// Mitsubishi GX Works2 project: A02_20260228_0   PLC: Q03UDV

TYPE Auto_Data : STRUCT
  X軸現在位置 : REAL;
  Y軸現在位置 : REAL;
END_STRUCT END_TYPE

// global labels: Global1
VAR_GLOBAL
  Auto_Data : Auto_Data;
  現在位置列 AT D400 : INT;
  現在位置層 AT D402 : INT;
END_VAR

// global labels: Coords
VAR_GLOBAL
  列座標 AT D3284 : ARRAY [1..14] OF REAL;
  層座標 AT D3274 : ARRAY [1..5] OF REAL;
  Z座標 AT D3270 : ARRAY [1..2] OF REAL;
END_VAR

PROGRAM 09  // Alram
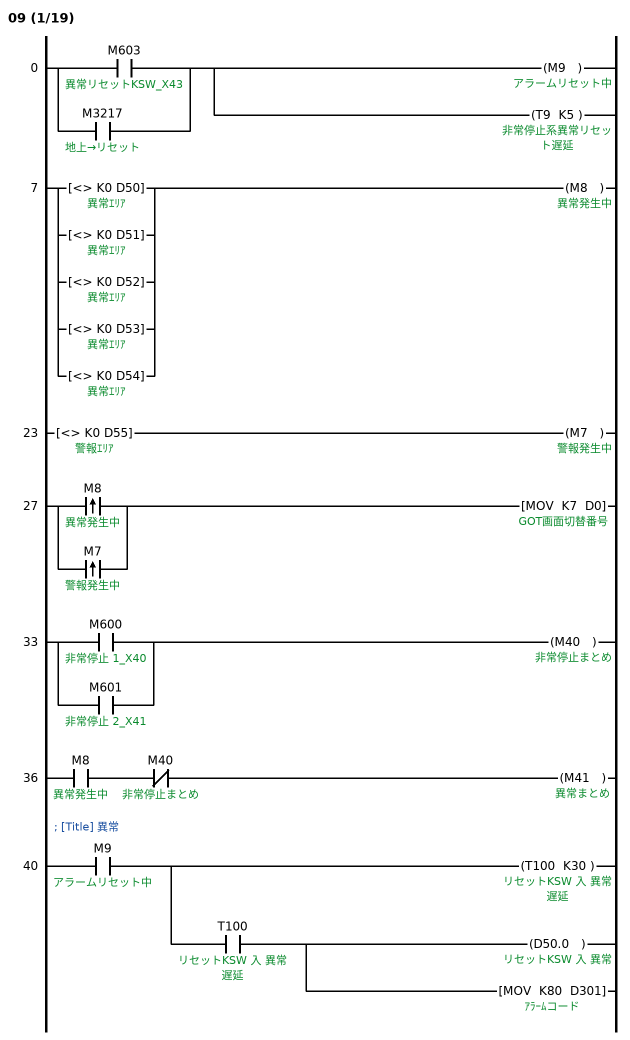
0     LD      M603  ; 異常リセットKSW_X43
      OR      M3217  ; 地上→リセット
      OUT     M9  ; アラームリセット中
      OUT     T9 K5  ; 非常停止系異常リセット遅延
7     LD<>    K0 D50  ; 異常ｴﾘｱ
      OR<>    K0 D51  ; 異常ｴﾘｱ
      OR<>    K0 D52  ; 異常ｴﾘｱ
      OR<>    K0 D53  ; 異常ｴﾘｱ
      OR<>    K0 D54  ; 異常ｴﾘｱ
      OUT     M8  ; 異常発生中
23    LD<>    K0 D55  ; 警報ｴﾘｱ
      OUT     M7  ; 警報発生中
27    LDP     M8  ; 異常発生中
      ORP     M7  ; 警報発生中
      MOV     K7 D0  ; GOT画面切替番号
33    LD      M600  ; 非常停止 1_X40
      OR      M601  ; 非常停止 2_X41
      OUT     M40  ; 非常停止まとめ
36    LD      M8  ; 異常発生中
      ANI     M40  ; 非常停止まとめ
      OUT     M41  ; 異常まとめ
; [Title] 異常
40    LD      M9  ; アラームリセット中
      OUT     T100 K30  ; リセットKSW 入 異常 遅延
      AND     T100  ; リセットKSW 入 異常 遅延
      OUT     D50.0  ; リセットKSW 入 異常
      MOV     K80 D301  ; ｱﾗｰﾑコード
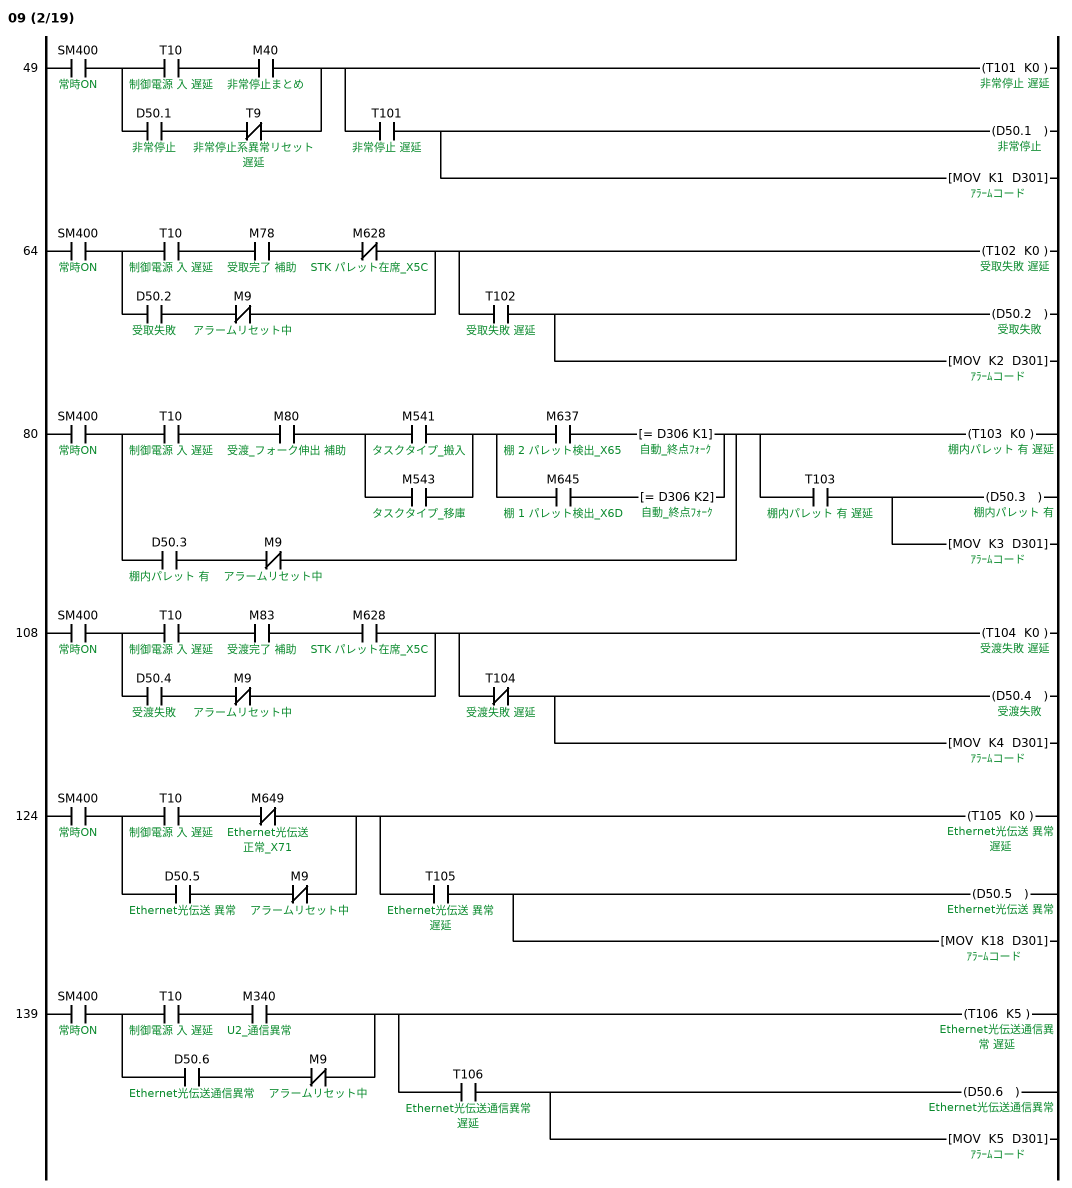
49    LD      SM400  ; 常時ON
      LD      T10  ; 制御電源 入 遅延
      AND     M40  ; 非常停止まとめ
      LD      D50.1  ; 非常停止
      ANI     T9  ; 非常停止系異常リセット遅延
      ORB
      ANB
      OUT     T101 K0  ; 非常停止 遅延
      AND     T101  ; 非常停止 遅延
      OUT     D50.1  ; 非常停止
      MOV     K1 D301
64    LD      SM400  ; 常時ON
      LD      T10  ; 制御電源 入 遅延
      AND     M78  ; 受取完了 補助
      ANI     M628  ; STK パレット在席_X5C
      LD      D50.2  ; 受取失敗
      ANI     M9  ; アラームリセット中
      ORB
      ANB
      OUT     T102 K0  ; 受取失敗 遅延
      AND     T102  ; 受取失敗 遅延
      OUT     D50.2  ; 受取失敗
      MOV     K2 D301
80    LD      SM400  ; 常時ON
      LD      T10  ; 制御電源 入 遅延
      AND     M80  ; 受渡_フォーク伸出 補助
      LD      M541  ; タスクタイプ_搬入
      OR      M543  ; タスクタイプ_移庫
      ANB
      LD      M637  ; 棚 2 パレット検出_X65
      AND=    D306 K1  ; 自動_終点ﾌｫｰｸ
      LD      M645  ; 棚 1 パレット検出_X6D
      AND=    D306 K2  ; 自動_終点ﾌｫｰｸ
      ORB
      ANB
      LD      D50.3  ; 棚内パレット 有
      ANI     M9  ; アラームリセット中
      ORB
      ANB
      OUT     T103 K0  ; 棚内パレット 有 遅延
      AND     T103  ; 棚内パレット 有 遅延
      OUT     D50.3  ; 棚内パレット 有
      MOV     K3 D301
108   LD      SM400  ; 常時ON
      LD      T10  ; 制御電源 入 遅延
      AND     M83  ; 受渡完了 補助
      AND     M628  ; STK パレット在席_X5C
      LD      D50.4  ; 受渡失敗
      ANI     M9  ; アラームリセット中
      ORB
      ANB
      OUT     T104 K0  ; 受渡失敗 遅延
      ANI     T104  ; 受渡失敗 遅延
      OUT     D50.4  ; 受渡失敗
      MOV     K4 D301
124   LD      SM400  ; 常時ON
      LD      T10  ; 制御電源 入 遅延
      ANI     M649  ; Ethernet光伝送 正常_X71
      LD      D50.5  ; Ethernet光伝送 異常
      ANI     M9  ; アラームリセット中
      ORB
      ANB
      OUT     T105 K0  ; Ethernet光伝送 異常 遅延
      AND     T105  ; Ethernet光伝送 異常 遅延
      OUT     D50.5  ; Ethernet光伝送 異常
      MOV     K18 D301
139   LD      SM400  ; 常時ON
      LD      T10  ; 制御電源 入 遅延
      AND     M340  ; U2_通信異常
      LD      D50.6  ; Ethernet光伝送通信異常
      ANI     M9  ; アラームリセット中
      ORB
      ANB
      OUT     T106 K5  ; Ethernet光伝送通信異常 遅延
      AND     T106  ; Ethernet光伝送通信異常 遅延
      OUT     D50.6  ; Ethernet光伝送通信異常
      MOV     K5 D301
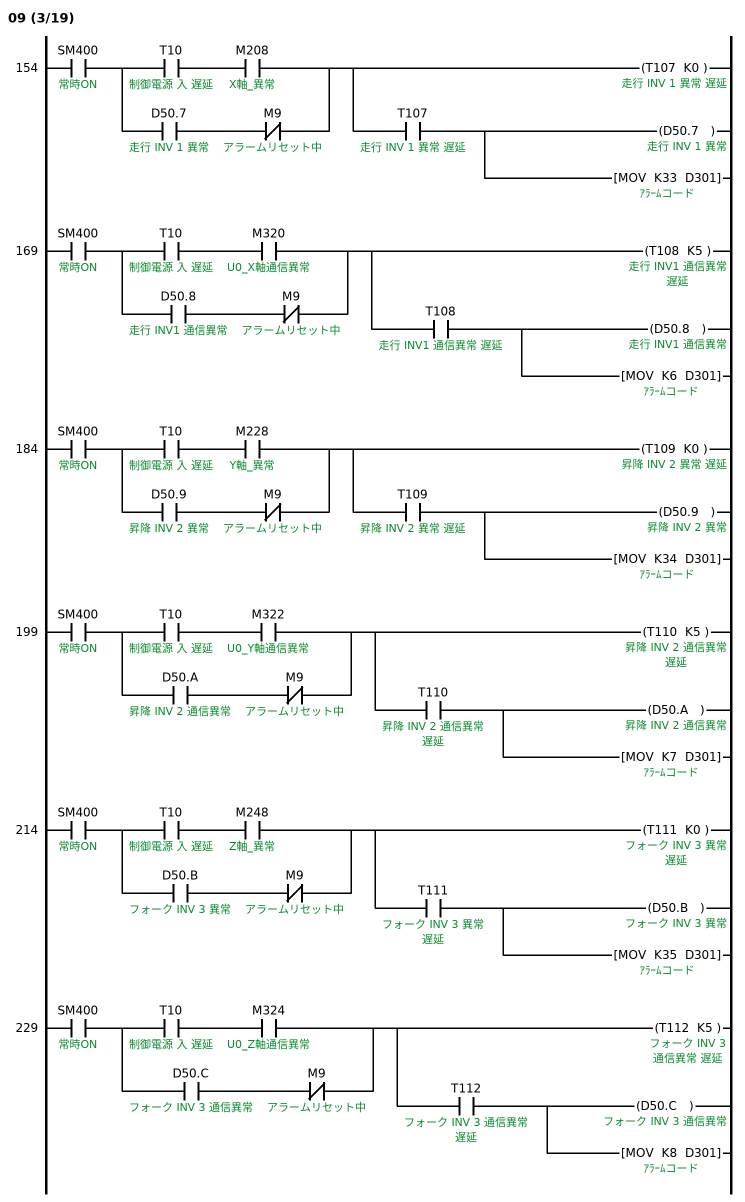
154   LD      SM400  ; 常時ON
      LD      T10  ; 制御電源 入 遅延
      AND     M208  ; X軸_異常
      LD      D50.7  ; 走行 INV 1 異常
      ANI     M9  ; アラームリセット中
      ORB
      ANB
      OUT     T107 K0  ; 走行 INV 1 異常 遅延
      AND     T107  ; 走行 INV 1 異常 遅延
      OUT     D50.7  ; 走行 INV 1 異常
      MOV     K33 D301
169   LD      SM400  ; 常時ON
      LD      T10  ; 制御電源 入 遅延
      AND     M320  ; U0_X軸通信異常
      LD      D50.8  ; 走行 INV1 通信異常
      ANI     M9  ; アラームリセット中
      ORB
      ANB
      OUT     T108 K5  ; 走行 INV1 通信異常 遅延
      AND     T108  ; 走行 INV1 通信異常 遅延
      OUT     D50.8  ; 走行 INV1 通信異常
      MOV     K6 D301
184   LD      SM400  ; 常時ON
      LD      T10  ; 制御電源 入 遅延
      AND     M228  ; Y軸_異常
      LD      D50.9  ; 昇降 INV 2 異常
      ANI     M9  ; アラームリセット中
      ORB
      ANB
      OUT     T109 K0  ; 昇降 INV 2 異常 遅延
      AND     T109  ; 昇降 INV 2 異常 遅延
      OUT     D50.9  ; 昇降 INV 2 異常
      MOV     K34 D301
199   LD      SM400  ; 常時ON
      LD      T10  ; 制御電源 入 遅延
      AND     M322  ; U0_Y軸通信異常
      LD      D50.A  ; 昇降 INV 2 通信異常
      ANI     M9  ; アラームリセット中
      ORB
      ANB
      OUT     T110 K5  ; 昇降 INV 2 通信異常 遅延
      AND     T110  ; 昇降 INV 2 通信異常 遅延
      OUT     D50.A  ; 昇降 INV 2 通信異常
      MOV     K7 D301
214   LD      SM400  ; 常時ON
      LD      T10  ; 制御電源 入 遅延
      AND     M248  ; Z軸_異常
      LD      D50.B  ; フォーク INV 3 異常
      ANI     M9  ; アラームリセット中
      ORB
      ANB
      OUT     T111 K0  ; フォーク INV 3 異常 遅延
      AND     T111  ; フォーク INV 3 異常 遅延
      OUT     D50.B  ; フォーク INV 3 異常
      MOV     K35 D301
229   LD      SM400  ; 常時ON
      LD      T10  ; 制御電源 入 遅延
      AND     M324  ; U0_Z軸通信異常
      LD      D50.C  ; フォーク INV 3 通信異常
      ANI     M9  ; アラームリセット中
      ORB
      ANB
      OUT     T112 K5  ; フォーク INV 3 通信異常 遅延
      AND     T112  ; フォーク INV 3 通信異常 遅延
      OUT     D50.C  ; フォーク INV 3 通信異常
      MOV     K8 D301
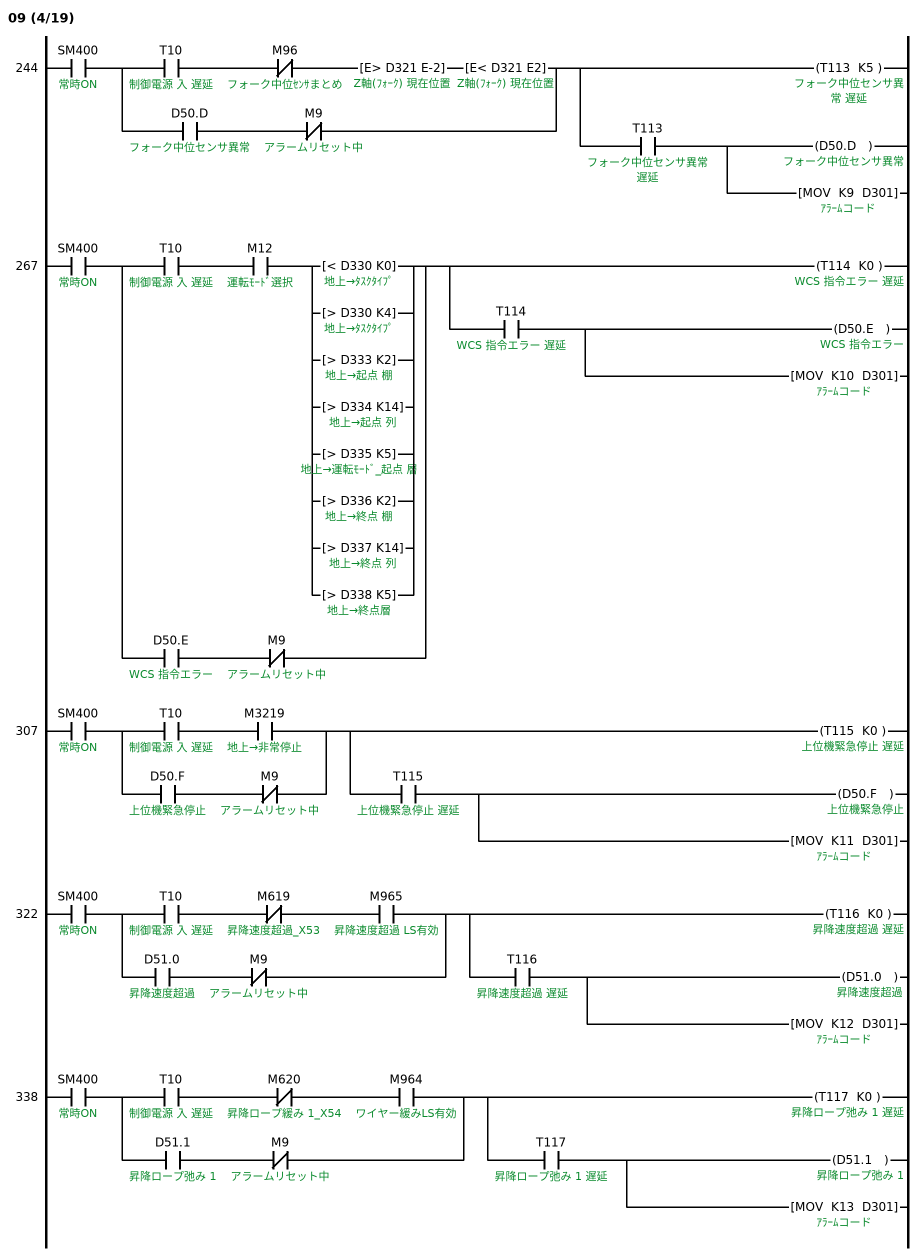
244   LD      SM400  ; 常時ON
      LD      T10  ; 制御電源 入 遅延
      ANI     M96  ; フォーク中位ｾﾝｻまとめ
      ANDE>   D321 E-2  ; Z軸(ﾌｫｰｸ) 現在位置
      ANDE<   D321 E2  ; Z軸(ﾌｫｰｸ) 現在位置
      LD      D50.D  ; フォーク中位センサ異常
      ANI     M9  ; アラームリセット中
      ORB
      ANB
      OUT     T113 K5  ; フォーク中位センサ異常 遅延
      AND     T113  ; フォーク中位センサ異常 遅延
      OUT     D50.D  ; フォーク中位センサ異常
      MOV     K9 D301
267   LD      SM400  ; 常時ON
      LD      T10  ; 制御電源 入 遅延
      AND     M12  ; 運転ﾓｰﾄﾞ選択
      LD<     D330 K0  ; 地上→ﾀｽｸﾀｲﾌﾟ
      OR>     D330 K4  ; 地上→ﾀｽｸﾀｲﾌﾟ
      OR>     D333 K2  ; 地上→起点 棚
      OR>     D334 K14  ; 地上→起点 列
      OR>     D335 K5  ; 地上→運転ﾓｰﾄﾞ_起点 層
      OR>     D336 K2  ; 地上→終点 棚
      OR>     D337 K14  ; 地上→終点 列
      OR>     D338 K5  ; 地上→終点層
      ANB
      LD      D50.E  ; WCS 指令エラー
      ANI     M9  ; アラームリセット中
      ORB
      ANB
      OUT     T114 K0  ; WCS 指令エラー 遅延
      AND     T114  ; WCS 指令エラー 遅延
      OUT     D50.E  ; WCS 指令エラー
      MOV     K10 D301
307   LD      SM400  ; 常時ON
      LD      T10  ; 制御電源 入 遅延
      AND     M3219  ; 地上→非常停止
      LD      D50.F  ; 上位機緊急停止
      ANI     M9  ; アラームリセット中
      ORB
      ANB
      OUT     T115 K0  ; 上位機緊急停止 遅延
      AND     T115  ; 上位機緊急停止 遅延
      OUT     D50.F  ; 上位機緊急停止
      MOV     K11 D301
322   LD      SM400  ; 常時ON
      LD      T10  ; 制御電源 入 遅延
      ANI     M619  ; 昇降速度超過_X53
      AND     M965  ; 昇降速度超過 LS有効
      LD      D51.0  ; 昇降速度超過
      ANI     M9  ; アラームリセット中
      ORB
      ANB
      OUT     T116 K0  ; 昇降速度超過 遅延
      AND     T116  ; 昇降速度超過 遅延
      OUT     D51.0  ; 昇降速度超過
      MOV     K12 D301
338   LD      SM400  ; 常時ON
      LD      T10  ; 制御電源 入 遅延
      ANI     M620  ; 昇降ロープ緩み 1_X54
      AND     M964  ; ワイヤー緩みLS有効
      LD      D51.1  ; 昇降ロープ弛み 1
      ANI     M9  ; アラームリセット中
      ORB
      ANB
      OUT     T117 K0  ; 昇降ロープ弛み 1 遅延
      AND     T117  ; 昇降ロープ弛み 1 遅延
      OUT     D51.1  ; 昇降ロープ弛み 1
      MOV     K13 D301
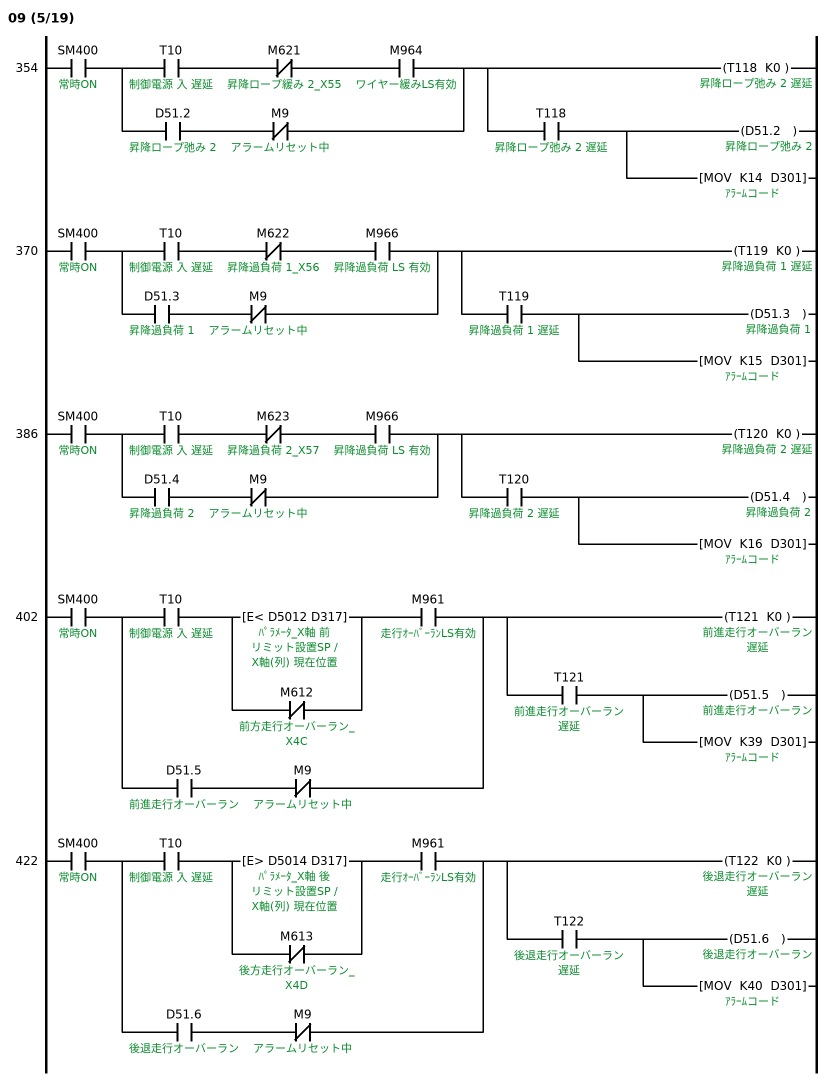
354   LD      SM400  ; 常時ON
      LD      T10  ; 制御電源 入 遅延
      ANI     M621  ; 昇降ロープ緩み 2_X55
      AND     M964  ; ワイヤー緩みLS有効
      LD      D51.2  ; 昇降ロープ弛み 2
      ANI     M9  ; アラームリセット中
      ORB
      ANB
      OUT     T118 K0  ; 昇降ロープ弛み 2 遅延
      AND     T118  ; 昇降ロープ弛み 2 遅延
      OUT     D51.2  ; 昇降ロープ弛み 2
      MOV     K14 D301
370   LD      SM400  ; 常時ON
      LD      T10  ; 制御電源 入 遅延
      ANI     M622  ; 昇降過負荷 1_X56
      AND     M966  ; 昇降過負荷 LS 有効
      LD      D51.3  ; 昇降過負荷 1
      ANI     M9  ; アラームリセット中
      ORB
      ANB
      OUT     T119 K0  ; 昇降過負荷 1 遅延
      AND     T119  ; 昇降過負荷 1 遅延
      OUT     D51.3  ; 昇降過負荷 1
      MOV     K15 D301
386   LD      SM400  ; 常時ON
      LD      T10  ; 制御電源 入 遅延
      ANI     M623  ; 昇降過負荷 2_X57
      AND     M966  ; 昇降過負荷 LS 有効
      LD      D51.4  ; 昇降過負荷 2
      ANI     M9  ; アラームリセット中
      ORB
      ANB
      OUT     T120 K0  ; 昇降過負荷 2 遅延
      AND     T120  ; 昇降過負荷 2 遅延
      OUT     D51.4  ; 昇降過負荷 2
      MOV     K16 D301
402   LD      SM400  ; 常時ON
      LD      T10  ; 制御電源 入 遅延
      LDE<    D5012 D317  ; ﾊﾟﾗﾒｰﾀ_X軸 前 リミット設置SP / X軸(列) 現在位置
      ORI     M612  ; 前方走行オーバーラン_X4C
      ANB
      AND     M961  ; 走行ｵｰﾊﾞｰﾗﾝLS有効
      LD      D51.5  ; 前進走行オーバーラン
      ANI     M9  ; アラームリセット中
      ORB
      ANB
      OUT     T121 K0  ; 前進走行オーバーラン 遅延
      AND     T121  ; 前進走行オーバーラン 遅延
      OUT     D51.5  ; 前進走行オーバーラン
      MOV     K39 D301
422   LD      SM400  ; 常時ON
      LD      T10  ; 制御電源 入 遅延
      LDE>    D5014 D317  ; ﾊﾟﾗﾒｰﾀ_X軸 後 リミット設置SP / X軸(列) 現在位置
      ORI     M613  ; 後方走行オーバーラン_X4D
      ANB
      AND     M961  ; 走行ｵｰﾊﾞｰﾗﾝLS有効
      LD      D51.6  ; 後退走行オーバーラン
      ANI     M9  ; アラームリセット中
      ORB
      ANB
      OUT     T122 K0  ; 後退走行オーバーラン 遅延
      AND     T122  ; 後退走行オーバーラン 遅延
      OUT     D51.6  ; 後退走行オーバーラン
      MOV     K40 D301
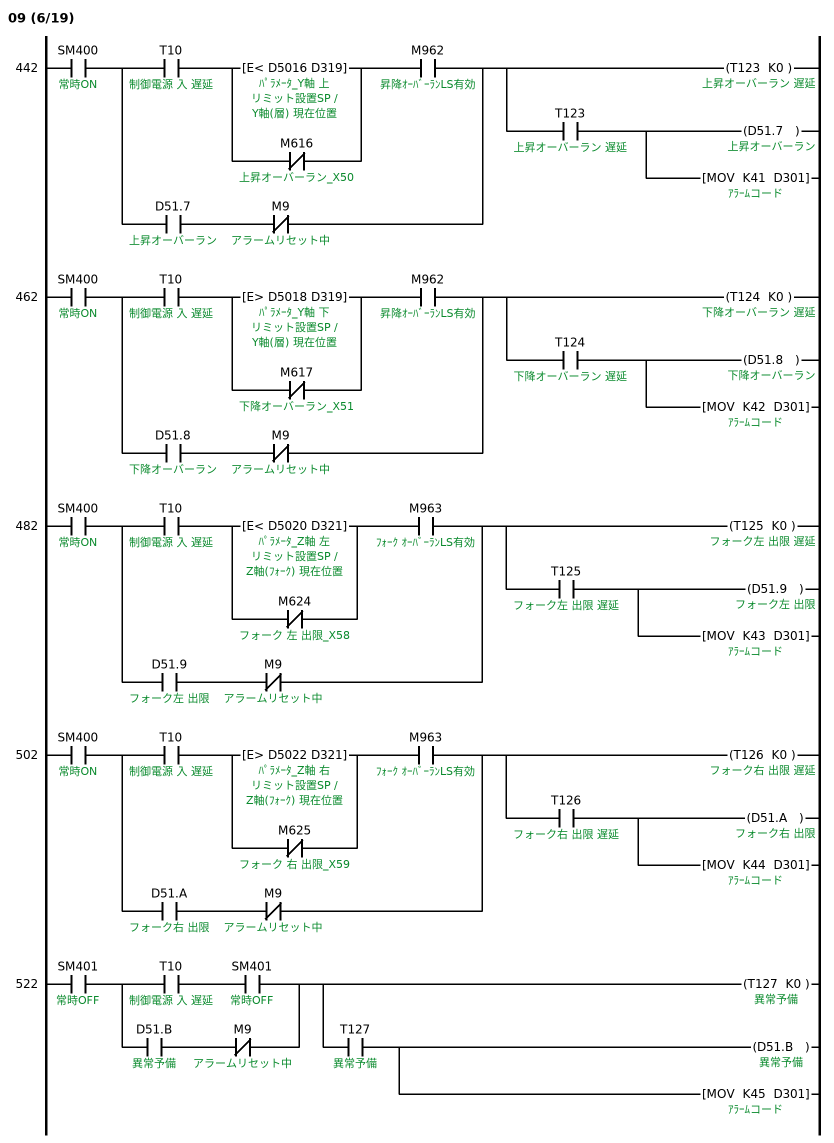
442   LD      SM400  ; 常時ON
      LD      T10  ; 制御電源 入 遅延
      LDE<    D5016 D319  ; ﾊﾟﾗﾒｰﾀ_Y軸 上 リミット設置SP / Y軸(層) 現在位置
      ORI     M616  ; 上昇オーバーラン_X50
      ANB
      AND     M962  ; 昇降ｵｰﾊﾞｰﾗﾝLS有効
      LD      D51.7  ; 上昇オーバーラン
      ANI     M9  ; アラームリセット中
      ORB
      ANB
      OUT     T123 K0  ; 上昇オーバーラン 遅延
      AND     T123  ; 上昇オーバーラン 遅延
      OUT     D51.7  ; 上昇オーバーラン
      MOV     K41 D301
462   LD      SM400  ; 常時ON
      LD      T10  ; 制御電源 入 遅延
      LDE>    D5018 D319  ; ﾊﾟﾗﾒｰﾀ_Y軸 下 リミット設置SP / Y軸(層) 現在位置
      ORI     M617  ; 下降オーバーラン_X51
      ANB
      AND     M962  ; 昇降ｵｰﾊﾞｰﾗﾝLS有効
      LD      D51.8  ; 下降オーバーラン
      ANI     M9  ; アラームリセット中
      ORB
      ANB
      OUT     T124 K0  ; 下降オーバーラン 遅延
      AND     T124  ; 下降オーバーラン 遅延
      OUT     D51.8  ; 下降オーバーラン
      MOV     K42 D301
482   LD      SM400  ; 常時ON
      LD      T10  ; 制御電源 入 遅延
      LDE<    D5020 D321  ; ﾊﾟﾗﾒｰﾀ_Z軸 左 リミット設置SP / Z軸(ﾌｫｰｸ) 現在位置
      ORI     M624  ; フォーク 左 出限_X58
      ANB
      AND     M963  ; ﾌｫｰｸ ｵｰﾊﾞｰﾗﾝLS有効
      LD      D51.9  ; フォーク左 出限
      ANI     M9  ; アラームリセット中
      ORB
      ANB
      OUT     T125 K0  ; フォーク左 出限 遅延
      AND     T125  ; フォーク左 出限 遅延
      OUT     D51.9  ; フォーク左 出限
      MOV     K43 D301
502   LD      SM400  ; 常時ON
      LD      T10  ; 制御電源 入 遅延
      LDE>    D5022 D321  ; ﾊﾟﾗﾒｰﾀ_Z軸 右 リミット設置SP / Z軸(ﾌｫｰｸ) 現在位置
      ORI     M625  ; フォーク 右 出限_X59
      ANB
      AND     M963  ; ﾌｫｰｸ ｵｰﾊﾞｰﾗﾝLS有効
      LD      D51.A  ; フォーク右 出限
      ANI     M9  ; アラームリセット中
      ORB
      ANB
      OUT     T126 K0  ; フォーク右 出限 遅延
      AND     T126  ; フォーク右 出限 遅延
      OUT     D51.A  ; フォーク右 出限
      MOV     K44 D301
522   LD      SM401  ; 常時OFF
      LD      T10  ; 制御電源 入 遅延
      AND     SM401  ; 常時OFF
      LD      D51.B  ; 異常予備
      ANI     M9  ; アラームリセット中
      ORB
      ANB
      OUT     T127 K0  ; 異常予備
      AND     T127  ; 異常予備
      OUT     D51.B  ; 異常予備
      MOV     K45 D301
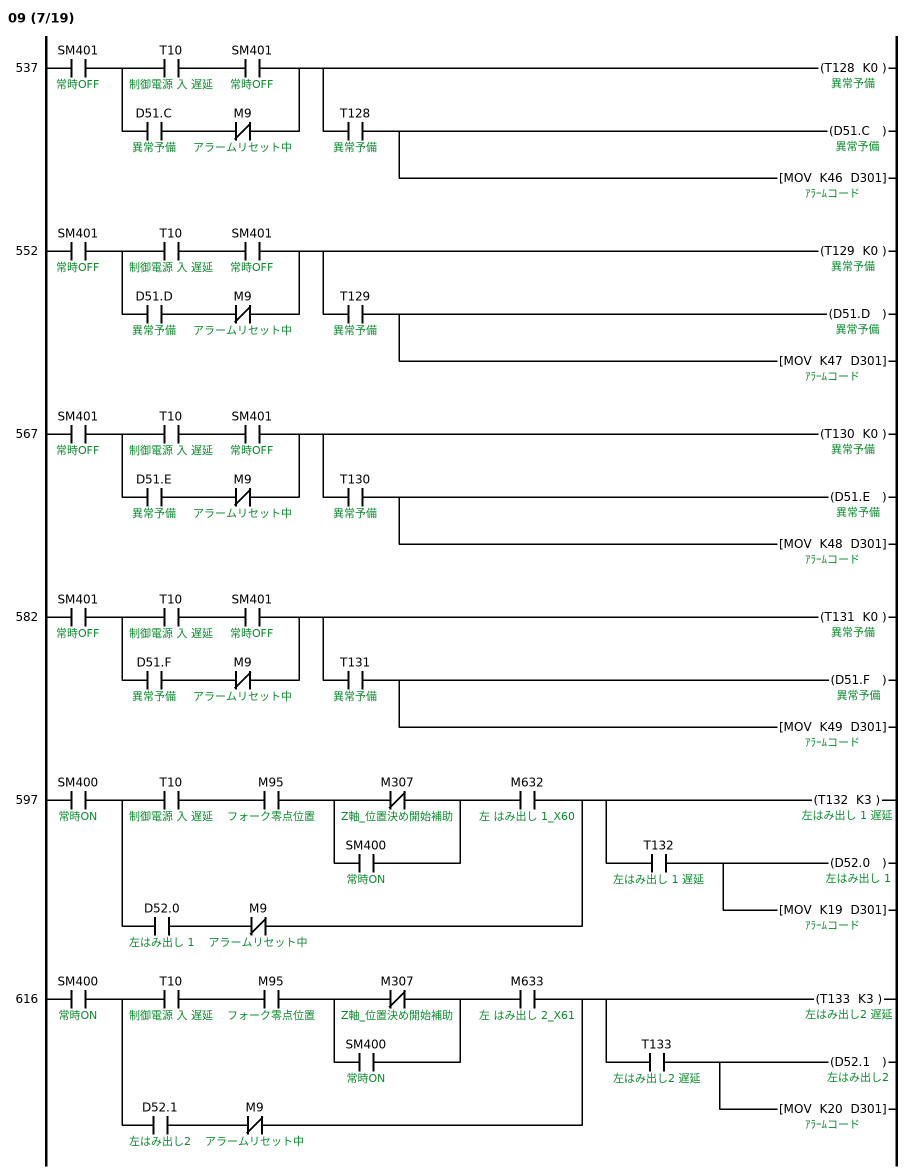
537   LD      SM401  ; 常時OFF
      LD      T10  ; 制御電源 入 遅延
      AND     SM401  ; 常時OFF
      LD      D51.C  ; 異常予備
      ANI     M9  ; アラームリセット中
      ORB
      ANB
      OUT     T128 K0  ; 異常予備
      AND     T128  ; 異常予備
      OUT     D51.C  ; 異常予備
      MOV     K46 D301
552   LD      SM401  ; 常時OFF
      LD      T10  ; 制御電源 入 遅延
      AND     SM401  ; 常時OFF
      LD      D51.D  ; 異常予備
      ANI     M9  ; アラームリセット中
      ORB
      ANB
      OUT     T129 K0  ; 異常予備
      AND     T129  ; 異常予備
      OUT     D51.D  ; 異常予備
      MOV     K47 D301
567   LD      SM401  ; 常時OFF
      LD      T10  ; 制御電源 入 遅延
      AND     SM401  ; 常時OFF
      LD      D51.E  ; 異常予備
      ANI     M9  ; アラームリセット中
      ORB
      ANB
      OUT     T130 K0  ; 異常予備
      AND     T130  ; 異常予備
      OUT     D51.E  ; 異常予備
      MOV     K48 D301
582   LD      SM401  ; 常時OFF
      LD      T10  ; 制御電源 入 遅延
      AND     SM401  ; 常時OFF
      LD      D51.F  ; 異常予備
      ANI     M9  ; アラームリセット中
      ORB
      ANB
      OUT     T131 K0  ; 異常予備
      AND     T131  ; 異常予備
      OUT     D51.F  ; 異常予備
      MOV     K49 D301
597   LD      SM400  ; 常時ON
      LD      T10  ; 制御電源 入 遅延
      AND     M95  ; フォーク零点位置
      LDI     M307  ; Z軸_位置決め開始補助
      OR      SM400  ; 常時ON
      ANB
      AND     M632  ; 左 はみ出し 1_X60
      LD      D52.0  ; 左はみ出し 1
      ANI     M9  ; アラームリセット中
      ORB
      ANB
      OUT     T132 K3  ; 左はみ出し 1 遅延
      AND     T132  ; 左はみ出し 1 遅延
      OUT     D52.0  ; 左はみ出し 1
      MOV     K19 D301
616   LD      SM400  ; 常時ON
      LD      T10  ; 制御電源 入 遅延
      AND     M95  ; フォーク零点位置
      LDI     M307  ; Z軸_位置決め開始補助
      OR      SM400  ; 常時ON
      ANB
      AND     M633  ; 左 はみ出し 2_X61
      LD      D52.1  ; 左はみ出し2
      ANI     M9  ; アラームリセット中
      ORB
      ANB
      OUT     T133 K3  ; 左はみ出し2 遅延
      AND     T133  ; 左はみ出し2 遅延
      OUT     D52.1  ; 左はみ出し2
      MOV     K20 D301
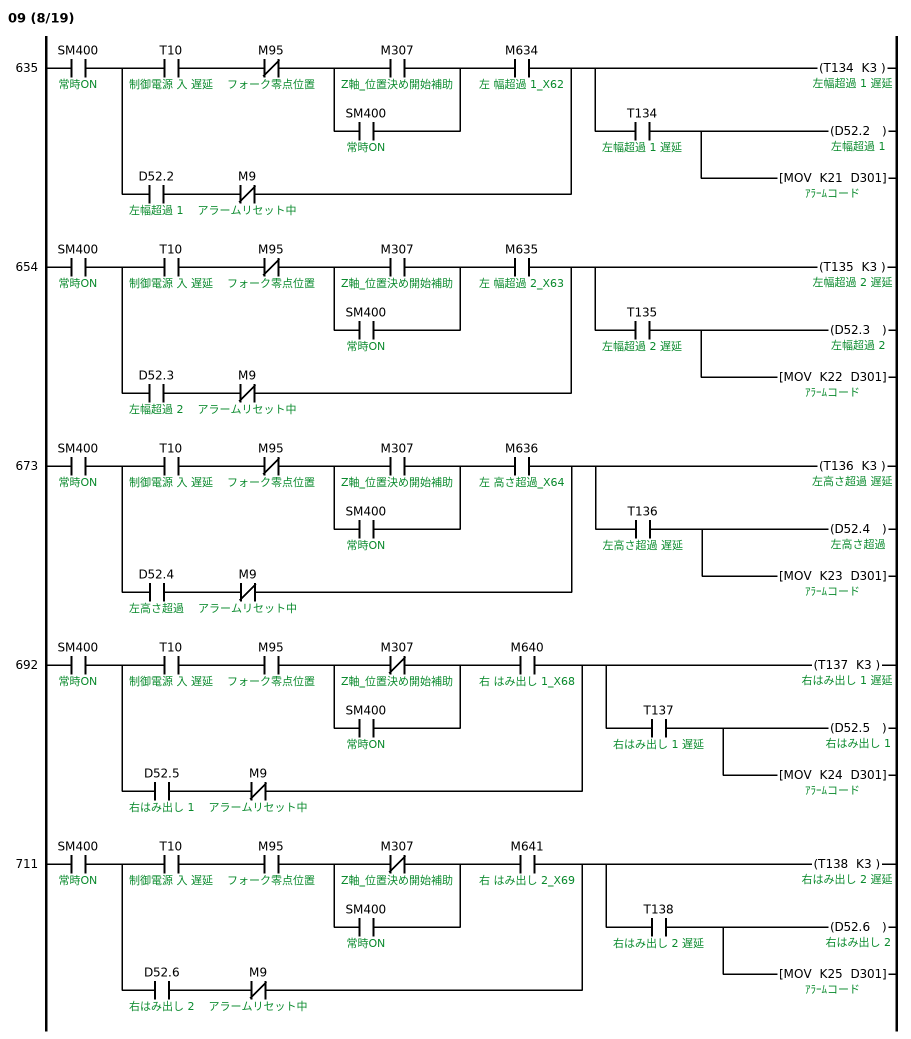
635   LD      SM400  ; 常時ON
      LD      T10  ; 制御電源 入 遅延
      ANI     M95  ; フォーク零点位置
      LD      M307  ; Z軸_位置決め開始補助
      OR      SM400  ; 常時ON
      ANB
      AND     M634  ; 左 幅超過 1_X62
      LD      D52.2  ; 左幅超過 1
      ANI     M9  ; アラームリセット中
      ORB
      ANB
      OUT     T134 K3  ; 左幅超過 1 遅延
      AND     T134  ; 左幅超過 1 遅延
      OUT     D52.2  ; 左幅超過 1
      MOV     K21 D301
654   LD      SM400  ; 常時ON
      LD      T10  ; 制御電源 入 遅延
      ANI     M95  ; フォーク零点位置
      LD      M307  ; Z軸_位置決め開始補助
      OR      SM400  ; 常時ON
      ANB
      AND     M635  ; 左 幅超過 2_X63
      LD      D52.3  ; 左幅超過 2
      ANI     M9  ; アラームリセット中
      ORB
      ANB
      OUT     T135 K3  ; 左幅超過 2 遅延
      AND     T135  ; 左幅超過 2 遅延
      OUT     D52.3  ; 左幅超過 2
      MOV     K22 D301
673   LD      SM400  ; 常時ON
      LD      T10  ; 制御電源 入 遅延
      ANI     M95  ; フォーク零点位置
      LD      M307  ; Z軸_位置決め開始補助
      OR      SM400  ; 常時ON
      ANB
      AND     M636  ; 左 高さ超過_X64
      LD      D52.4  ; 左高さ超過
      ANI     M9  ; アラームリセット中
      ORB
      ANB
      OUT     T136 K3  ; 左高さ超過 遅延
      AND     T136  ; 左高さ超過 遅延
      OUT     D52.4  ; 左高さ超過
      MOV     K23 D301
692   LD      SM400  ; 常時ON
      LD      T10  ; 制御電源 入 遅延
      AND     M95  ; フォーク零点位置
      LDI     M307  ; Z軸_位置決め開始補助
      OR      SM400  ; 常時ON
      ANB
      AND     M640  ; 右 はみ出し 1_X68
      LD      D52.5  ; 右はみ出し 1
      ANI     M9  ; アラームリセット中
      ORB
      ANB
      OUT     T137 K3  ; 右はみ出し 1 遅延
      AND     T137  ; 右はみ出し 1 遅延
      OUT     D52.5  ; 右はみ出し 1
      MOV     K24 D301
711   LD      SM400  ; 常時ON
      LD      T10  ; 制御電源 入 遅延
      AND     M95  ; フォーク零点位置
      LDI     M307  ; Z軸_位置決め開始補助
      OR      SM400  ; 常時ON
      ANB
      AND     M641  ; 右 はみ出し 2_X69
      LD      D52.6  ; 右はみ出し 2
      ANI     M9  ; アラームリセット中
      ORB
      ANB
      OUT     T138 K3  ; 右はみ出し 2 遅延
      AND     T138  ; 右はみ出し 2 遅延
      OUT     D52.6  ; 右はみ出し 2
      MOV     K25 D301
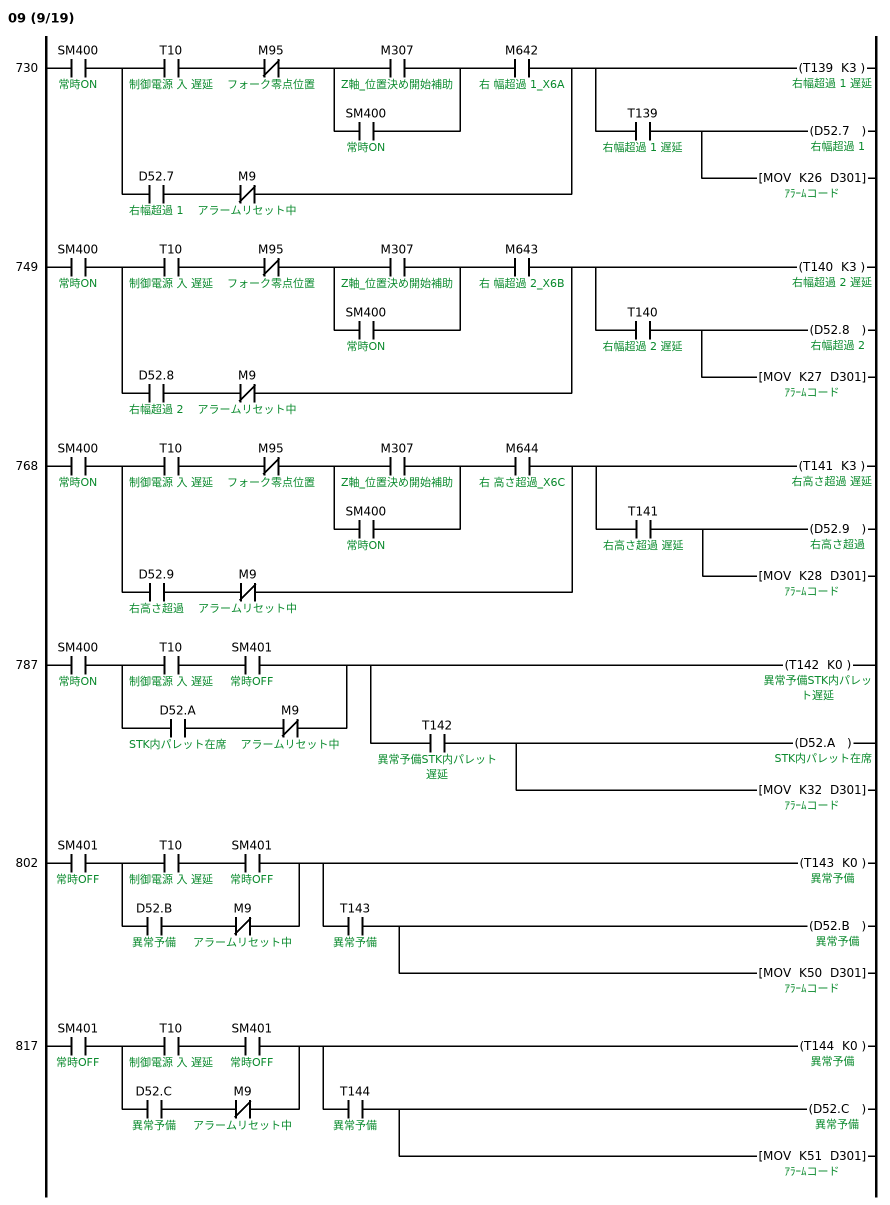
730   LD      SM400  ; 常時ON
      LD      T10  ; 制御電源 入 遅延
      ANI     M95  ; フォーク零点位置
      LD      M307  ; Z軸_位置決め開始補助
      OR      SM400  ; 常時ON
      ANB
      AND     M642  ; 右 幅超過 1_X6A
      LD      D52.7  ; 右幅超過 1
      ANI     M9  ; アラームリセット中
      ORB
      ANB
      OUT     T139 K3  ; 右幅超過 1 遅延
      AND     T139  ; 右幅超過 1 遅延
      OUT     D52.7  ; 右幅超過 1
      MOV     K26 D301
749   LD      SM400  ; 常時ON
      LD      T10  ; 制御電源 入 遅延
      ANI     M95  ; フォーク零点位置
      LD      M307  ; Z軸_位置決め開始補助
      OR      SM400  ; 常時ON
      ANB
      AND     M643  ; 右 幅超過 2_X6B
      LD      D52.8  ; 右幅超過 2
      ANI     M9  ; アラームリセット中
      ORB
      ANB
      OUT     T140 K3  ; 右幅超過 2 遅延
      AND     T140  ; 右幅超過 2 遅延
      OUT     D52.8  ; 右幅超過 2
      MOV     K27 D301
768   LD      SM400  ; 常時ON
      LD      T10  ; 制御電源 入 遅延
      ANI     M95  ; フォーク零点位置
      LD      M307  ; Z軸_位置決め開始補助
      OR      SM400  ; 常時ON
      ANB
      AND     M644  ; 右 高さ超過_X6C
      LD      D52.9  ; 右高さ超過
      ANI     M9  ; アラームリセット中
      ORB
      ANB
      OUT     T141 K3  ; 右高さ超過 遅延
      AND     T141  ; 右高さ超過 遅延
      OUT     D52.9  ; 右高さ超過
      MOV     K28 D301
787   LD      SM400  ; 常時ON
      LD      T10  ; 制御電源 入 遅延
      AND     SM401  ; 常時OFF
      LD      D52.A  ; STK内パレット在席
      ANI     M9  ; アラームリセット中
      ORB
      ANB
      OUT     T142 K0  ; 異常予備STK内パレット遅延
      AND     T142  ; 異常予備STK内パレット遅延
      OUT     D52.A  ; STK内パレット在席
      MOV     K32 D301
802   LD      SM401  ; 常時OFF
      LD      T10  ; 制御電源 入 遅延
      AND     SM401  ; 常時OFF
      LD      D52.B  ; 異常予備
      ANI     M9  ; アラームリセット中
      ORB
      ANB
      OUT     T143 K0  ; 異常予備
      AND     T143  ; 異常予備
      OUT     D52.B  ; 異常予備
      MOV     K50 D301
817   LD      SM401  ; 常時OFF
      LD      T10  ; 制御電源 入 遅延
      AND     SM401  ; 常時OFF
      LD      D52.C  ; 異常予備
      ANI     M9  ; アラームリセット中
      ORB
      ANB
      OUT     T144 K0  ; 異常予備
      AND     T144  ; 異常予備
      OUT     D52.C  ; 異常予備
      MOV     K51 D301
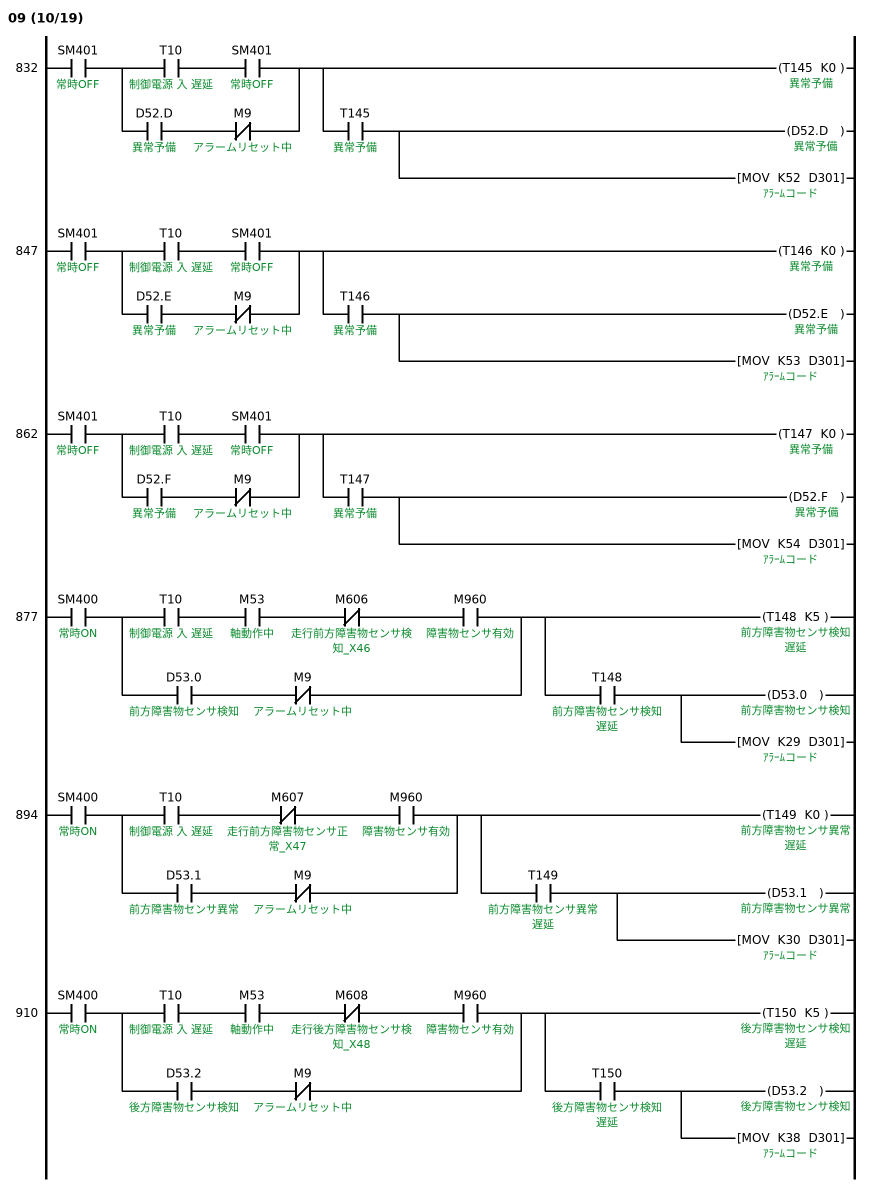
832   LD      SM401  ; 常時OFF
      LD      T10  ; 制御電源 入 遅延
      AND     SM401  ; 常時OFF
      LD      D52.D  ; 異常予備
      ANI     M9  ; アラームリセット中
      ORB
      ANB
      OUT     T145 K0  ; 異常予備
      AND     T145  ; 異常予備
      OUT     D52.D  ; 異常予備
      MOV     K52 D301
847   LD      SM401  ; 常時OFF
      LD      T10  ; 制御電源 入 遅延
      AND     SM401  ; 常時OFF
      LD      D52.E  ; 異常予備
      ANI     M9  ; アラームリセット中
      ORB
      ANB
      OUT     T146 K0  ; 異常予備
      AND     T146  ; 異常予備
      OUT     D52.E  ; 異常予備
      MOV     K53 D301
862   LD      SM401  ; 常時OFF
      LD      T10  ; 制御電源 入 遅延
      AND     SM401  ; 常時OFF
      LD      D52.F  ; 異常予備
      ANI     M9  ; アラームリセット中
      ORB
      ANB
      OUT     T147 K0  ; 異常予備
      AND     T147  ; 異常予備
      OUT     D52.F  ; 異常予備
      MOV     K54 D301
877   LD      SM400  ; 常時ON
      LD      T10  ; 制御電源 入 遅延
      AND     M53  ; 軸動作中
      ANI     M606  ; 走行前方障害物センサ検知_X46
      AND     M960  ; 障害物センサ有効
      LD      D53.0  ; 前方障害物センサ検知
      ANI     M9  ; アラームリセット中
      ORB
      ANB
      OUT     T148 K5  ; 前方障害物センサ検知 遅延
      AND     T148  ; 前方障害物センサ検知 遅延
      OUT     D53.0  ; 前方障害物センサ検知
      MOV     K29 D301
894   LD      SM400  ; 常時ON
      LD      T10  ; 制御電源 入 遅延
      ANI     M607  ; 走行前方障害物センサ正常_X47
      AND     M960  ; 障害物センサ有効
      LD      D53.1  ; 前方障害物センサ異常
      ANI     M9  ; アラームリセット中
      ORB
      ANB
      OUT     T149 K0  ; 前方障害物センサ異常 遅延
      AND     T149  ; 前方障害物センサ異常 遅延
      OUT     D53.1  ; 前方障害物センサ異常
      MOV     K30 D301
910   LD      SM400  ; 常時ON
      LD      T10  ; 制御電源 入 遅延
      AND     M53  ; 軸動作中
      ANI     M608  ; 走行後方障害物センサ検知_X48
      AND     M960  ; 障害物センサ有効
      LD      D53.2  ; 後方障害物センサ検知
      ANI     M9  ; アラームリセット中
      ORB
      ANB
      OUT     T150 K5  ; 後方障害物センサ検知 遅延
      AND     T150  ; 後方障害物センサ検知 遅延
      OUT     D53.2  ; 後方障害物センサ検知
      MOV     K38 D301
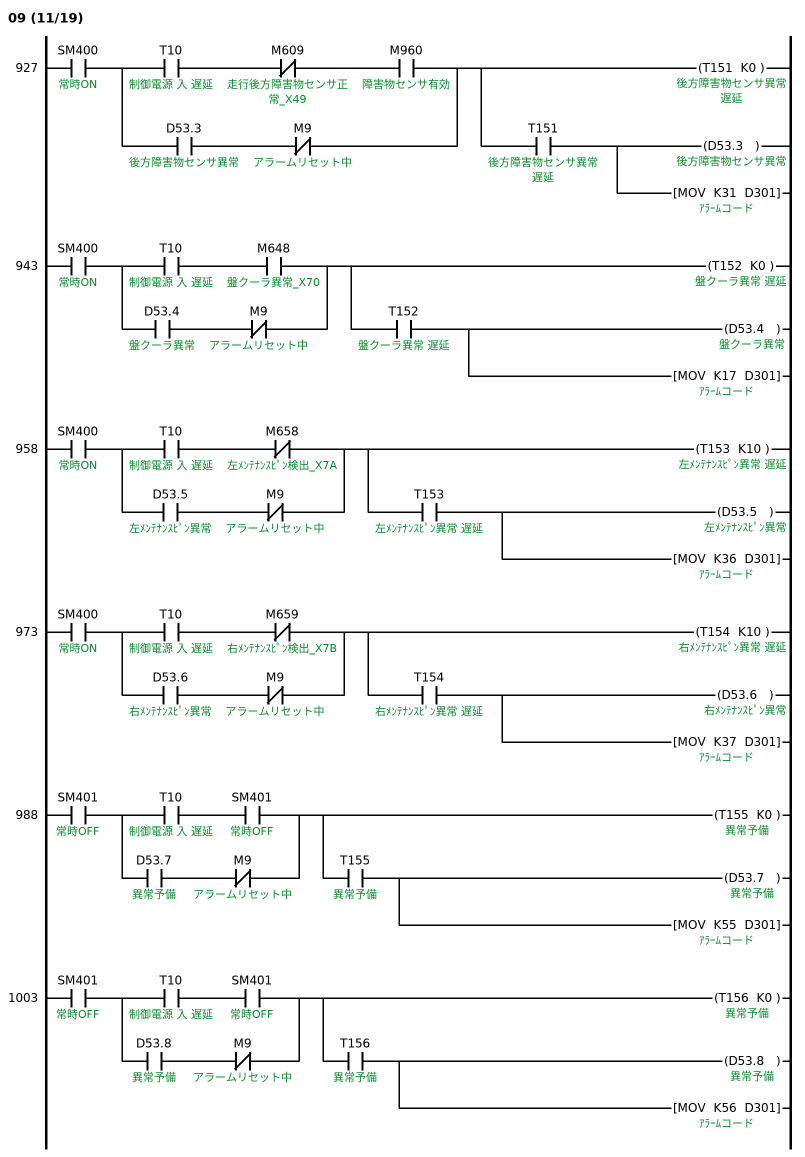
927   LD      SM400  ; 常時ON
      LD      T10  ; 制御電源 入 遅延
      ANI     M609  ; 走行後方障害物センサ正常_X49
      AND     M960  ; 障害物センサ有効
      LD      D53.3  ; 後方障害物センサ異常
      ANI     M9  ; アラームリセット中
      ORB
      ANB
      OUT     T151 K0  ; 後方障害物センサ異常 遅延
      AND     T151  ; 後方障害物センサ異常 遅延
      OUT     D53.3  ; 後方障害物センサ異常
      MOV     K31 D301
943   LD      SM400  ; 常時ON
      LD      T10  ; 制御電源 入 遅延
      AND     M648  ; 盤クーラ異常_X70
      LD      D53.4  ; 盤クーラ異常
      ANI     M9  ; アラームリセット中
      ORB
      ANB
      OUT     T152 K0  ; 盤クーラ異常 遅延
      AND     T152  ; 盤クーラ異常 遅延
      OUT     D53.4  ; 盤クーラ異常
      MOV     K17 D301
958   LD      SM400  ; 常時ON
      LD      T10  ; 制御電源 入 遅延
      ANI     M658  ; 左ﾒﾝﾃﾅﾝｽﾋﾟﾝ検出_X7A
      LD      D53.5  ; 左ﾒﾝﾃﾅﾝｽﾋﾟﾝ異常
      ANI     M9  ; アラームリセット中
      ORB
      ANB
      OUT     T153 K10  ; 左ﾒﾝﾃﾅﾝｽﾋﾟﾝ異常 遅延
      AND     T153  ; 左ﾒﾝﾃﾅﾝｽﾋﾟﾝ異常 遅延
      OUT     D53.5  ; 左ﾒﾝﾃﾅﾝｽﾋﾟﾝ異常
      MOV     K36 D301
973   LD      SM400  ; 常時ON
      LD      T10  ; 制御電源 入 遅延
      ANI     M659  ; 右ﾒﾝﾃﾅﾝｽﾋﾟﾝ検出_X7B
      LD      D53.6  ; 右ﾒﾝﾃﾅﾝｽﾋﾟﾝ異常
      ANI     M9  ; アラームリセット中
      ORB
      ANB
      OUT     T154 K10  ; 右ﾒﾝﾃﾅﾝｽﾋﾟﾝ異常 遅延
      AND     T154  ; 右ﾒﾝﾃﾅﾝｽﾋﾟﾝ異常 遅延
      OUT     D53.6  ; 右ﾒﾝﾃﾅﾝｽﾋﾟﾝ異常
      MOV     K37 D301
988   LD      SM401  ; 常時OFF
      LD      T10  ; 制御電源 入 遅延
      AND     SM401  ; 常時OFF
      LD      D53.7  ; 異常予備
      ANI     M9  ; アラームリセット中
      ORB
      ANB
      OUT     T155 K0  ; 異常予備
      AND     T155  ; 異常予備
      OUT     D53.7  ; 異常予備
      MOV     K55 D301
1003  LD      SM401  ; 常時OFF
      LD      T10  ; 制御電源 入 遅延
      AND     SM401  ; 常時OFF
      LD      D53.8  ; 異常予備
      ANI     M9  ; アラームリセット中
      ORB
      ANB
      OUT     T156 K0  ; 異常予備
      AND     T156  ; 異常予備
      OUT     D53.8  ; 異常予備
      MOV     K56 D301
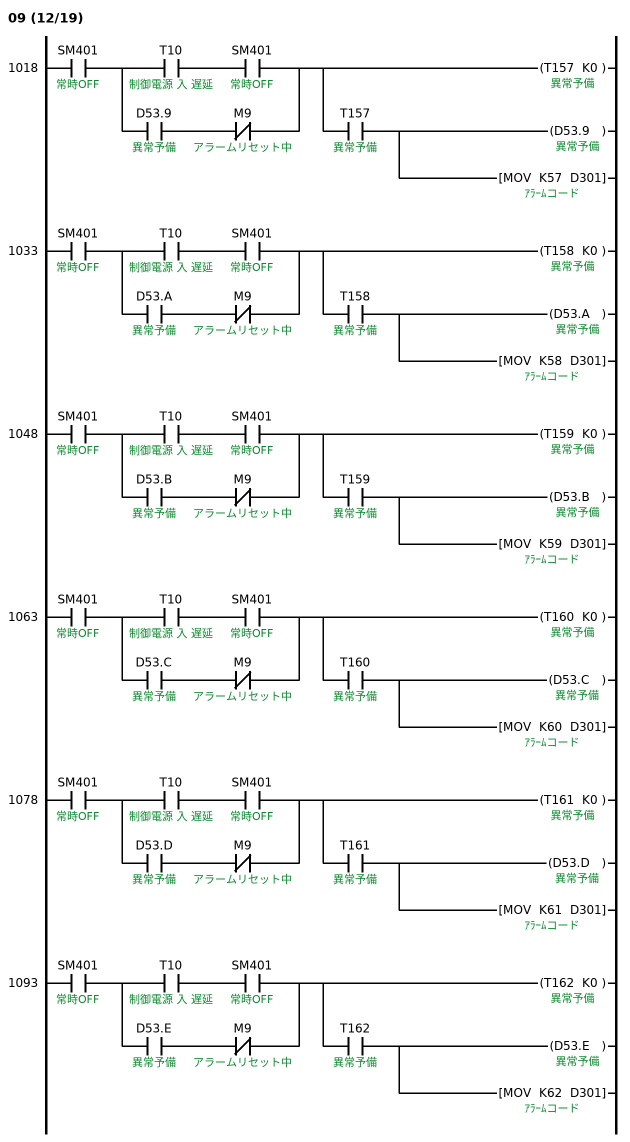
1018  LD      SM401  ; 常時OFF
      LD      T10  ; 制御電源 入 遅延
      AND     SM401  ; 常時OFF
      LD      D53.9  ; 異常予備
      ANI     M9  ; アラームリセット中
      ORB
      ANB
      OUT     T157 K0  ; 異常予備
      AND     T157  ; 異常予備
      OUT     D53.9  ; 異常予備
      MOV     K57 D301
1033  LD      SM401  ; 常時OFF
      LD      T10  ; 制御電源 入 遅延
      AND     SM401  ; 常時OFF
      LD      D53.A  ; 異常予備
      ANI     M9  ; アラームリセット中
      ORB
      ANB
      OUT     T158 K0  ; 異常予備
      AND     T158  ; 異常予備
      OUT     D53.A  ; 異常予備
      MOV     K58 D301
1048  LD      SM401  ; 常時OFF
      LD      T10  ; 制御電源 入 遅延
      AND     SM401  ; 常時OFF
      LD      D53.B  ; 異常予備
      ANI     M9  ; アラームリセット中
      ORB
      ANB
      OUT     T159 K0  ; 異常予備
      AND     T159  ; 異常予備
      OUT     D53.B  ; 異常予備
      MOV     K59 D301
1063  LD      SM401  ; 常時OFF
      LD      T10  ; 制御電源 入 遅延
      AND     SM401  ; 常時OFF
      LD      D53.C  ; 異常予備
      ANI     M9  ; アラームリセット中
      ORB
      ANB
      OUT     T160 K0  ; 異常予備
      AND     T160  ; 異常予備
      OUT     D53.C  ; 異常予備
      MOV     K60 D301
1078  LD      SM401  ; 常時OFF
      LD      T10  ; 制御電源 入 遅延
      AND     SM401  ; 常時OFF
      LD      D53.D  ; 異常予備
      ANI     M9  ; アラームリセット中
      ORB
      ANB
      OUT     T161 K0  ; 異常予備
      AND     T161  ; 異常予備
      OUT     D53.D  ; 異常予備
      MOV     K61 D301
1093  LD      SM401  ; 常時OFF
      LD      T10  ; 制御電源 入 遅延
      AND     SM401  ; 常時OFF
      LD      D53.E  ; 異常予備
      ANI     M9  ; アラームリセット中
      ORB
      ANB
      OUT     T162 K0  ; 異常予備
      AND     T162  ; 異常予備
      OUT     D53.E  ; 異常予備
      MOV     K62 D301
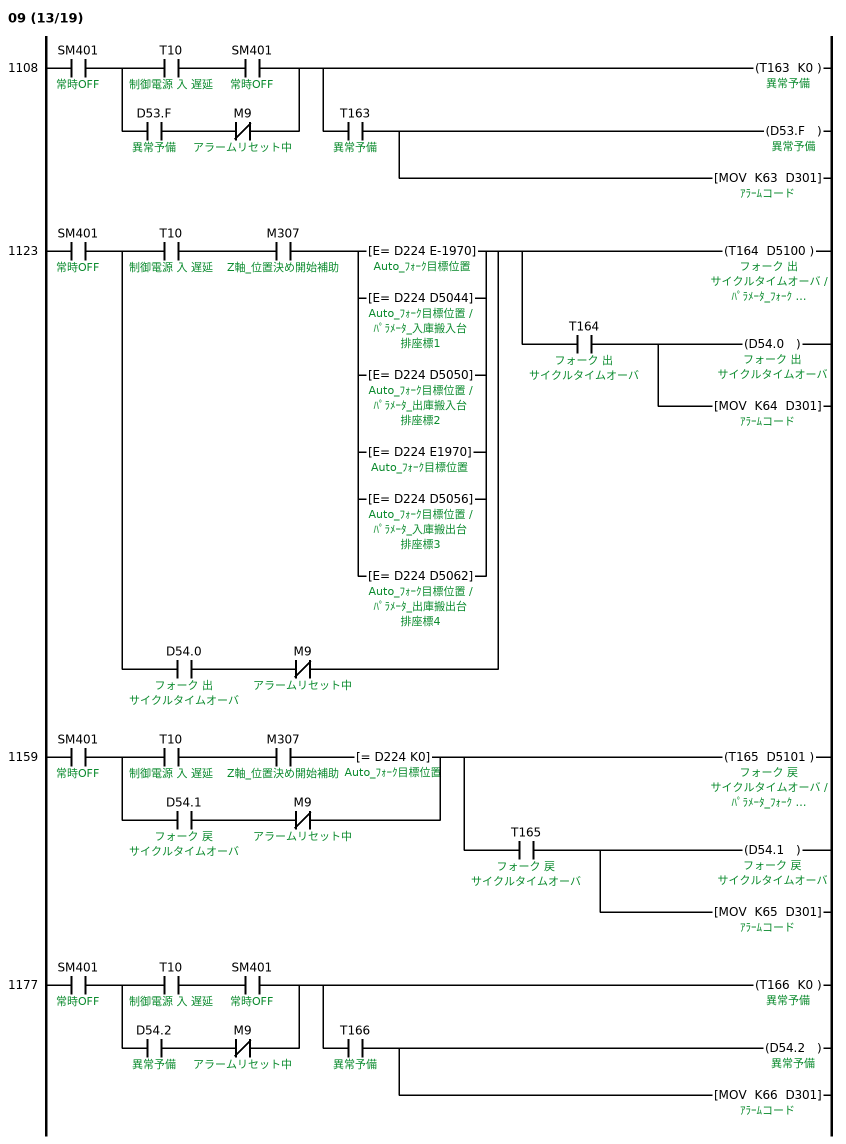
1108  LD      SM401  ; 常時OFF
      LD      T10  ; 制御電源 入 遅延
      AND     SM401  ; 常時OFF
      LD      D53.F  ; 異常予備
      ANI     M9  ; アラームリセット中
      ORB
      ANB
      OUT     T163 K0  ; 異常予備
      AND     T163  ; 異常予備
      OUT     D53.F  ; 異常予備
      MOV     K63 D301
1123  LD      SM401  ; 常時OFF
      LD      T10  ; 制御電源 入 遅延
      AND     M307  ; Z軸_位置決め開始補助
      LDE=    D224 E-1970  ; Auto_ﾌｫｰｸ目標位置
      ORE=    D224 D5044  ; Auto_ﾌｫｰｸ目標位置 / ﾊﾟﾗﾒｰﾀ_入庫搬入台  排座標1
      ORE=    D224 D5050  ; Auto_ﾌｫｰｸ目標位置 / ﾊﾟﾗﾒｰﾀ_出庫搬入台  排座標2
      ORE=    D224 E1970  ; Auto_ﾌｫｰｸ目標位置
      ORE=    D224 D5056  ; Auto_ﾌｫｰｸ目標位置 / ﾊﾟﾗﾒｰﾀ_入庫搬出台  排座標3
      ORE=    D224 D5062  ; Auto_ﾌｫｰｸ目標位置 / ﾊﾟﾗﾒｰﾀ_出庫搬出台  排座標4
      ANB
      LD      D54.0  ; フォーク 出 サイクルタイムオーバ
      ANI     M9  ; アラームリセット中
      ORB
      ANB
      OUT     T164 D5100  ; フォーク 出 サイクルタイムオーバ / ﾊﾟﾗﾒｰﾀ_ﾌｫｰｸ 出 ｻｲｸﾙﾀｲﾑｵｰﾊﾞｰ
      AND     T164  ; フォーク 出 サイクルタイムオーバ
      OUT     D54.0  ; フォーク 出 サイクルタイムオーバ
      MOV     K64 D301
1159  LD      SM401  ; 常時OFF
      LD      T10  ; 制御電源 入 遅延
      AND     M307  ; Z軸_位置決め開始補助
      AND=    D224 K0  ; Auto_ﾌｫｰｸ目標位置
      LD      D54.1  ; フォーク 戻 サイクルタイムオーバ
      ANI     M9  ; アラームリセット中
      ORB
      ANB
      OUT     T165 D5101  ; フォーク 戻 サイクルタイムオーバ / ﾊﾟﾗﾒｰﾀ_ﾌｫｰｸ 戻 ｻｲｸﾙﾀｲﾑｵｰﾊﾞｰ
      AND     T165  ; フォーク 戻 サイクルタイムオーバ
      OUT     D54.1  ; フォーク 戻 サイクルタイムオーバ
      MOV     K65 D301
1177  LD      SM401  ; 常時OFF
      LD      T10  ; 制御電源 入 遅延
      AND     SM401  ; 常時OFF
      LD      D54.2  ; 異常予備
      ANI     M9  ; アラームリセット中
      ORB
      ANB
      OUT     T166 K0  ; 異常予備
      AND     T166  ; 異常予備
      OUT     D54.2  ; 異常予備
      MOV     K66 D301
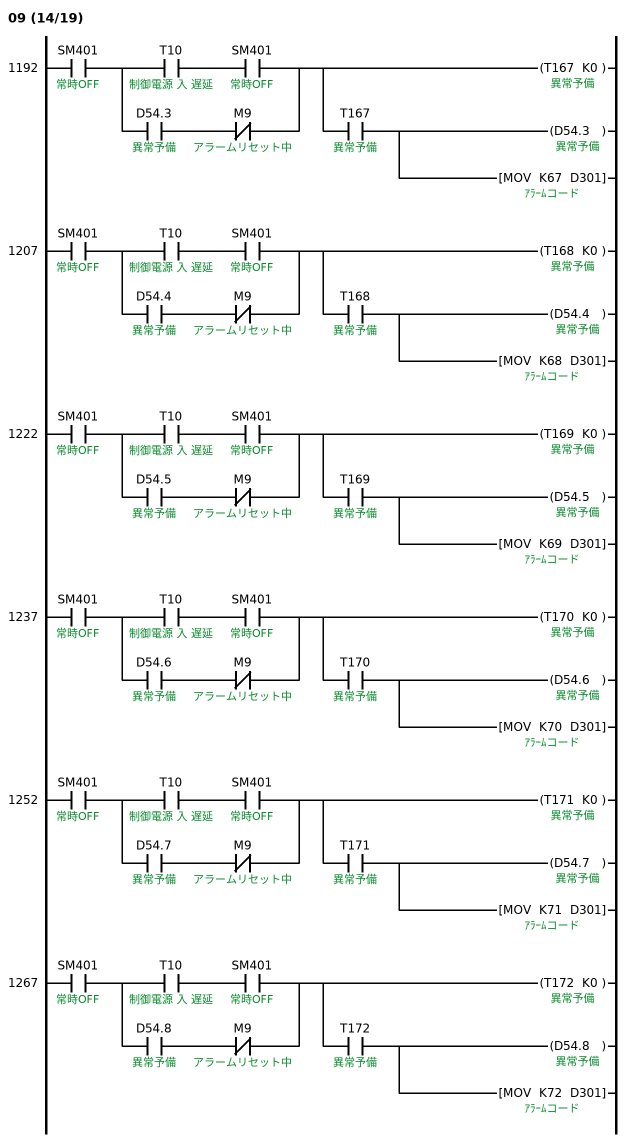
1192  LD      SM401  ; 常時OFF
      LD      T10  ; 制御電源 入 遅延
      AND     SM401  ; 常時OFF
      LD      D54.3  ; 異常予備
      ANI     M9  ; アラームリセット中
      ORB
      ANB
      OUT     T167 K0  ; 異常予備
      AND     T167  ; 異常予備
      OUT     D54.3  ; 異常予備
      MOV     K67 D301
1207  LD      SM401  ; 常時OFF
      LD      T10  ; 制御電源 入 遅延
      AND     SM401  ; 常時OFF
      LD      D54.4  ; 異常予備
      ANI     M9  ; アラームリセット中
      ORB
      ANB
      OUT     T168 K0  ; 異常予備
      AND     T168  ; 異常予備
      OUT     D54.4  ; 異常予備
      MOV     K68 D301
1222  LD      SM401  ; 常時OFF
      LD      T10  ; 制御電源 入 遅延
      AND     SM401  ; 常時OFF
      LD      D54.5  ; 異常予備
      ANI     M9  ; アラームリセット中
      ORB
      ANB
      OUT     T169 K0  ; 異常予備
      AND     T169  ; 異常予備
      OUT     D54.5  ; 異常予備
      MOV     K69 D301
1237  LD      SM401  ; 常時OFF
      LD      T10  ; 制御電源 入 遅延
      AND     SM401  ; 常時OFF
      LD      D54.6  ; 異常予備
      ANI     M9  ; アラームリセット中
      ORB
      ANB
      OUT     T170 K0  ; 異常予備
      AND     T170  ; 異常予備
      OUT     D54.6  ; 異常予備
      MOV     K70 D301
1252  LD      SM401  ; 常時OFF
      LD      T10  ; 制御電源 入 遅延
      AND     SM401  ; 常時OFF
      LD      D54.7  ; 異常予備
      ANI     M9  ; アラームリセット中
      ORB
      ANB
      OUT     T171 K0  ; 異常予備
      AND     T171  ; 異常予備
      OUT     D54.7  ; 異常予備
      MOV     K71 D301
1267  LD      SM401  ; 常時OFF
      LD      T10  ; 制御電源 入 遅延
      AND     SM401  ; 常時OFF
      LD      D54.8  ; 異常予備
      ANI     M9  ; アラームリセット中
      ORB
      ANB
      OUT     T172 K0  ; 異常予備
      AND     T172  ; 異常予備
      OUT     D54.8  ; 異常予備
      MOV     K72 D301
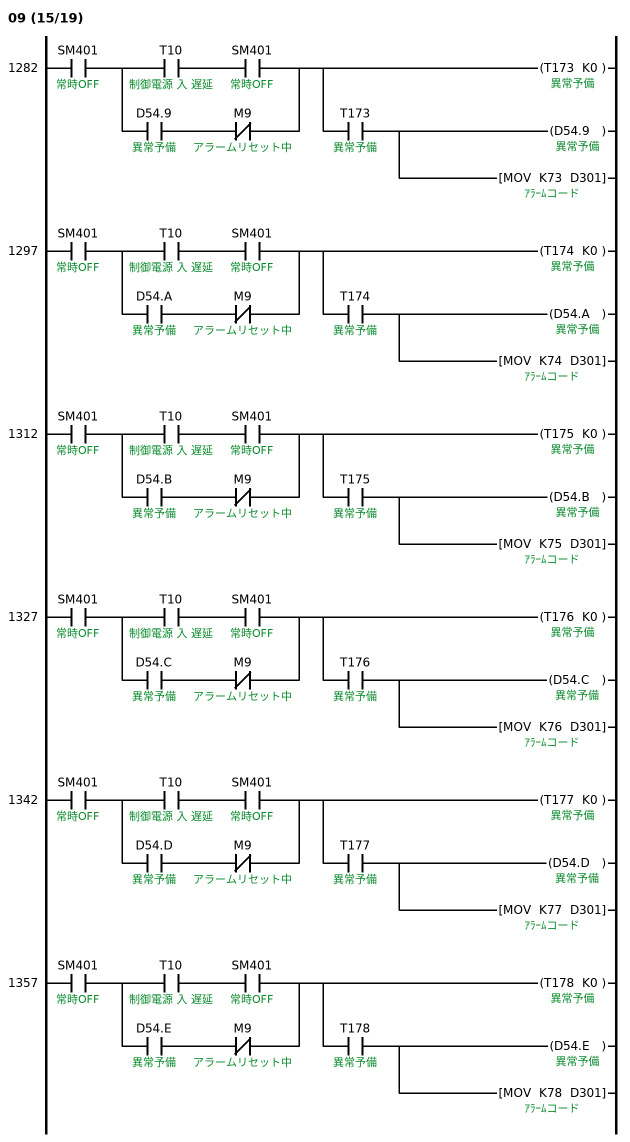
1282  LD      SM401  ; 常時OFF
      LD      T10  ; 制御電源 入 遅延
      AND     SM401  ; 常時OFF
      LD      D54.9  ; 異常予備
      ANI     M9  ; アラームリセット中
      ORB
      ANB
      OUT     T173 K0  ; 異常予備
      AND     T173  ; 異常予備
      OUT     D54.9  ; 異常予備
      MOV     K73 D301
1297  LD      SM401  ; 常時OFF
      LD      T10  ; 制御電源 入 遅延
      AND     SM401  ; 常時OFF
      LD      D54.A  ; 異常予備
      ANI     M9  ; アラームリセット中
      ORB
      ANB
      OUT     T174 K0  ; 異常予備
      AND     T174  ; 異常予備
      OUT     D54.A  ; 異常予備
      MOV     K74 D301
1312  LD      SM401  ; 常時OFF
      LD      T10  ; 制御電源 入 遅延
      AND     SM401  ; 常時OFF
      LD      D54.B  ; 異常予備
      ANI     M9  ; アラームリセット中
      ORB
      ANB
      OUT     T175 K0  ; 異常予備
      AND     T175  ; 異常予備
      OUT     D54.B  ; 異常予備
      MOV     K75 D301
1327  LD      SM401  ; 常時OFF
      LD      T10  ; 制御電源 入 遅延
      AND     SM401  ; 常時OFF
      LD      D54.C  ; 異常予備
      ANI     M9  ; アラームリセット中
      ORB
      ANB
      OUT     T176 K0  ; 異常予備
      AND     T176  ; 異常予備
      OUT     D54.C  ; 異常予備
      MOV     K76 D301
1342  LD      SM401  ; 常時OFF
      LD      T10  ; 制御電源 入 遅延
      AND     SM401  ; 常時OFF
      LD      D54.D  ; 異常予備
      ANI     M9  ; アラームリセット中
      ORB
      ANB
      OUT     T177 K0  ; 異常予備
      AND     T177  ; 異常予備
      OUT     D54.D  ; 異常予備
      MOV     K77 D301
1357  LD      SM401  ; 常時OFF
      LD      T10  ; 制御電源 入 遅延
      AND     SM401  ; 常時OFF
      LD      D54.E  ; 異常予備
      ANI     M9  ; アラームリセット中
      ORB
      ANB
      OUT     T178 K0  ; 異常予備
      AND     T178  ; 異常予備
      OUT     D54.E  ; 異常予備
      MOV     K78 D301
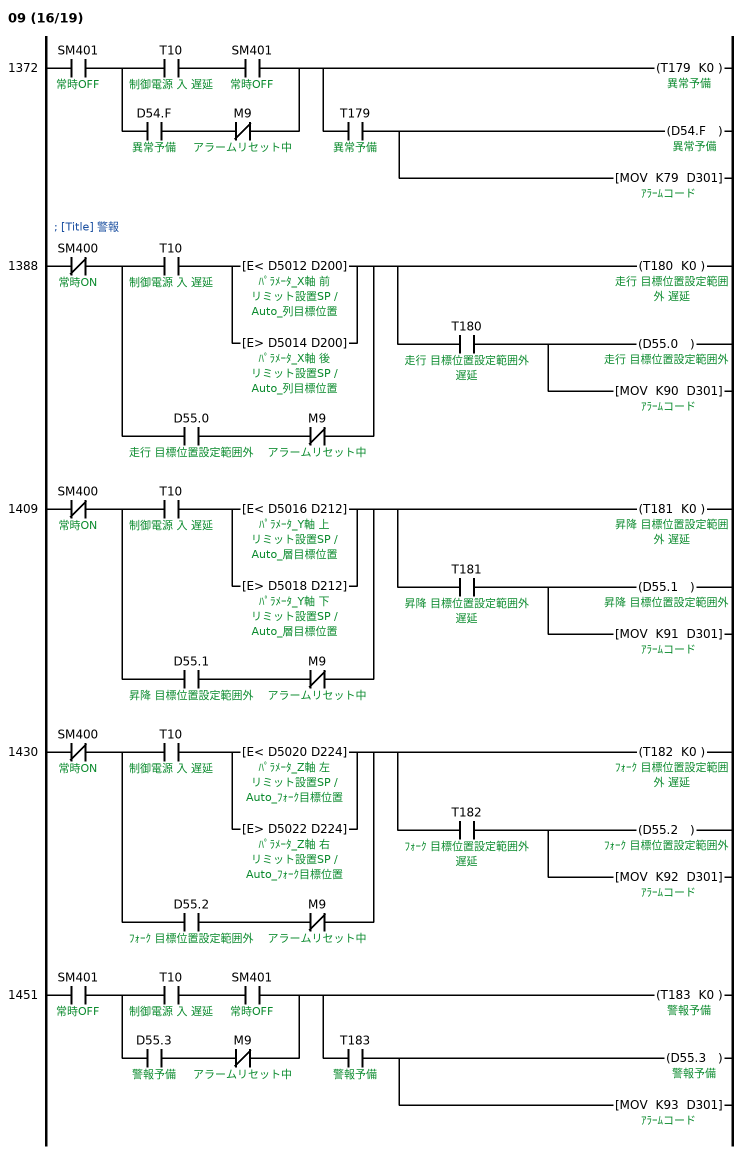
1372  LD      SM401  ; 常時OFF
      LD      T10  ; 制御電源 入 遅延
      AND     SM401  ; 常時OFF
      LD      D54.F  ; 異常予備
      ANI     M9  ; アラームリセット中
      ORB
      ANB
      OUT     T179 K0  ; 異常予備
      AND     T179  ; 異常予備
      OUT     D54.F  ; 異常予備
      MOV     K79 D301
; [Title] 警報
1388  LDI     SM400  ; 常時ON
      LD      T10  ; 制御電源 入 遅延
      LDE<    D5012 D200  ; ﾊﾟﾗﾒｰﾀ_X軸 前 リミット設置SP / Auto_列目標位置
      ORE>    D5014 D200  ; ﾊﾟﾗﾒｰﾀ_X軸 後 リミット設置SP / Auto_列目標位置
      ANB
      LD      D55.0  ; 走行 目標位置設定範囲外
      ANI     M9  ; アラームリセット中
      ORB
      ANB
      OUT     T180 K0  ; 走行 目標位置設定範囲外 遅延
      AND     T180  ; 走行 目標位置設定範囲外 遅延
      OUT     D55.0  ; 走行 目標位置設定範囲外
      MOV     K90 D301
1409  LDI     SM400  ; 常時ON
      LD      T10  ; 制御電源 入 遅延
      LDE<    D5016 D212  ; ﾊﾟﾗﾒｰﾀ_Y軸 上 リミット設置SP / Auto_層目標位置
      ORE>    D5018 D212  ; ﾊﾟﾗﾒｰﾀ_Y軸 下 リミット設置SP / Auto_層目標位置
      ANB
      LD      D55.1  ; 昇降 目標位置設定範囲外
      ANI     M9  ; アラームリセット中
      ORB
      ANB
      OUT     T181 K0  ; 昇降 目標位置設定範囲外 遅延
      AND     T181  ; 昇降 目標位置設定範囲外 遅延
      OUT     D55.1  ; 昇降 目標位置設定範囲外
      MOV     K91 D301
1430  LDI     SM400  ; 常時ON
      LD      T10  ; 制御電源 入 遅延
      LDE<    D5020 D224  ; ﾊﾟﾗﾒｰﾀ_Z軸 左 リミット設置SP / Auto_ﾌｫｰｸ目標位置
      ORE>    D5022 D224  ; ﾊﾟﾗﾒｰﾀ_Z軸 右 リミット設置SP / Auto_ﾌｫｰｸ目標位置
      ANB
      LD      D55.2  ; ﾌｫｰｸ 目標位置設定範囲外
      ANI     M9  ; アラームリセット中
      ORB
      ANB
      OUT     T182 K0  ; ﾌｫｰｸ 目標位置設定範囲外 遅延
      AND     T182  ; ﾌｫｰｸ 目標位置設定範囲外 遅延
      OUT     D55.2  ; ﾌｫｰｸ 目標位置設定範囲外
      MOV     K92 D301
1451  LD      SM401  ; 常時OFF
      LD      T10  ; 制御電源 入 遅延
      AND     SM401  ; 常時OFF
      LD      D55.3  ; 警報予備
      ANI     M9  ; アラームリセット中
      ORB
      ANB
      OUT     T183 K0  ; 警報予備
      AND     T183  ; 警報予備
      OUT     D55.3  ; 警報予備
      MOV     K93 D301
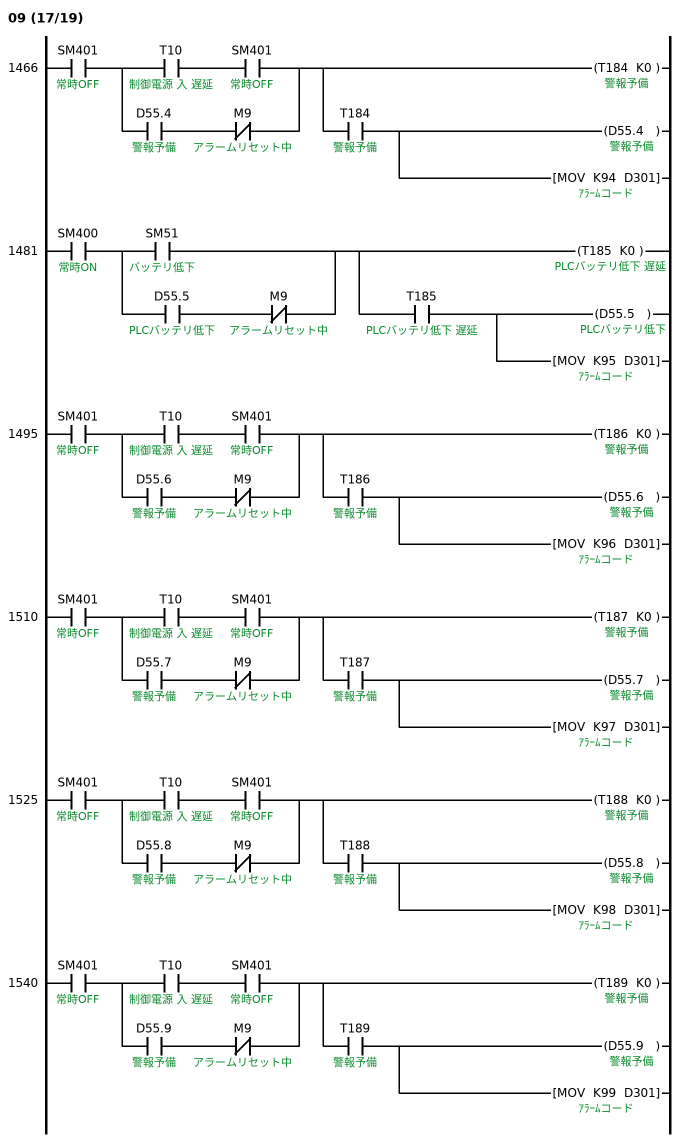
1466  LD      SM401  ; 常時OFF
      LD      T10  ; 制御電源 入 遅延
      AND     SM401  ; 常時OFF
      LD      D55.4  ; 警報予備
      ANI     M9  ; アラームリセット中
      ORB
      ANB
      OUT     T184 K0  ; 警報予備
      AND     T184  ; 警報予備
      OUT     D55.4  ; 警報予備
      MOV     K94 D301
1481  LD      SM400  ; 常時ON
      LD      SM51  ; バッテリ低下
      LD      D55.5  ; PLCバッテリ低下
      ANI     M9  ; アラームリセット中
      ORB
      ANB
      OUT     T185 K0  ; PLCバッテリ低下 遅延
      AND     T185  ; PLCバッテリ低下 遅延
      OUT     D55.5  ; PLCバッテリ低下
      MOV     K95 D301
1495  LD      SM401  ; 常時OFF
      LD      T10  ; 制御電源 入 遅延
      AND     SM401  ; 常時OFF
      LD      D55.6  ; 警報予備
      ANI     M9  ; アラームリセット中
      ORB
      ANB
      OUT     T186 K0  ; 警報予備
      AND     T186  ; 警報予備
      OUT     D55.6  ; 警報予備
      MOV     K96 D301
1510  LD      SM401  ; 常時OFF
      LD      T10  ; 制御電源 入 遅延
      AND     SM401  ; 常時OFF
      LD      D55.7  ; 警報予備
      ANI     M9  ; アラームリセット中
      ORB
      ANB
      OUT     T187 K0  ; 警報予備
      AND     T187  ; 警報予備
      OUT     D55.7  ; 警報予備
      MOV     K97 D301
1525  LD      SM401  ; 常時OFF
      LD      T10  ; 制御電源 入 遅延
      AND     SM401  ; 常時OFF
      LD      D55.8  ; 警報予備
      ANI     M9  ; アラームリセット中
      ORB
      ANB
      OUT     T188 K0  ; 警報予備
      AND     T188  ; 警報予備
      OUT     D55.8  ; 警報予備
      MOV     K98 D301
1540  LD      SM401  ; 常時OFF
      LD      T10  ; 制御電源 入 遅延
      AND     SM401  ; 常時OFF
      LD      D55.9  ; 警報予備
      ANI     M9  ; アラームリセット中
      ORB
      ANB
      OUT     T189 K0  ; 警報予備
      AND     T189  ; 警報予備
      OUT     D55.9  ; 警報予備
      MOV     K99 D301
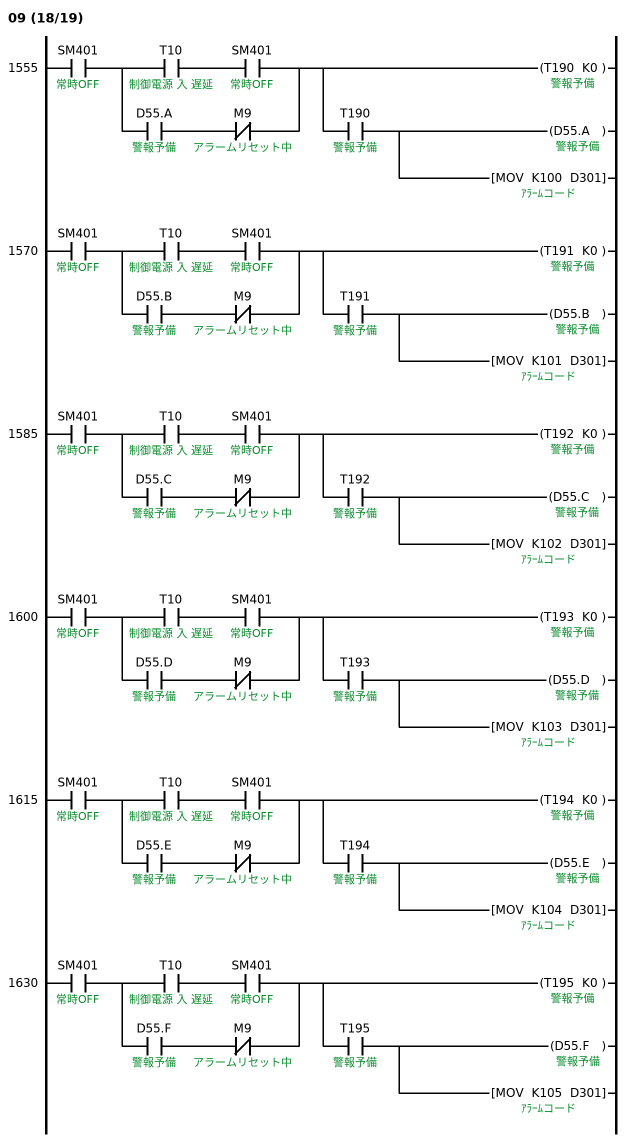
1555  LD      SM401  ; 常時OFF
      LD      T10  ; 制御電源 入 遅延
      AND     SM401  ; 常時OFF
      LD      D55.A  ; 警報予備
      ANI     M9  ; アラームリセット中
      ORB
      ANB
      OUT     T190 K0  ; 警報予備
      AND     T190  ; 警報予備
      OUT     D55.A  ; 警報予備
      MOV     K100 D301
1570  LD      SM401  ; 常時OFF
      LD      T10  ; 制御電源 入 遅延
      AND     SM401  ; 常時OFF
      LD      D55.B  ; 警報予備
      ANI     M9  ; アラームリセット中
      ORB
      ANB
      OUT     T191 K0  ; 警報予備
      AND     T191  ; 警報予備
      OUT     D55.B  ; 警報予備
      MOV     K101 D301
1585  LD      SM401  ; 常時OFF
      LD      T10  ; 制御電源 入 遅延
      AND     SM401  ; 常時OFF
      LD      D55.C  ; 警報予備
      ANI     M9  ; アラームリセット中
      ORB
      ANB
      OUT     T192 K0  ; 警報予備
      AND     T192  ; 警報予備
      OUT     D55.C  ; 警報予備
      MOV     K102 D301
1600  LD      SM401  ; 常時OFF
      LD      T10  ; 制御電源 入 遅延
      AND     SM401  ; 常時OFF
      LD      D55.D  ; 警報予備
      ANI     M9  ; アラームリセット中
      ORB
      ANB
      OUT     T193 K0  ; 警報予備
      AND     T193  ; 警報予備
      OUT     D55.D  ; 警報予備
      MOV     K103 D301
1615  LD      SM401  ; 常時OFF
      LD      T10  ; 制御電源 入 遅延
      AND     SM401  ; 常時OFF
      LD      D55.E  ; 警報予備
      ANI     M9  ; アラームリセット中
      ORB
      ANB
      OUT     T194 K0  ; 警報予備
      AND     T194  ; 警報予備
      OUT     D55.E  ; 警報予備
      MOV     K104 D301
1630  LD      SM401  ; 常時OFF
      LD      T10  ; 制御電源 入 遅延
      AND     SM401  ; 常時OFF
      LD      D55.F  ; 警報予備
      ANI     M9  ; アラームリセット中
      ORB
      ANB
      OUT     T195 K0  ; 警報予備
      AND     T195  ; 警報予備
      OUT     D55.F  ; 警報予備
      MOV     K105 D301
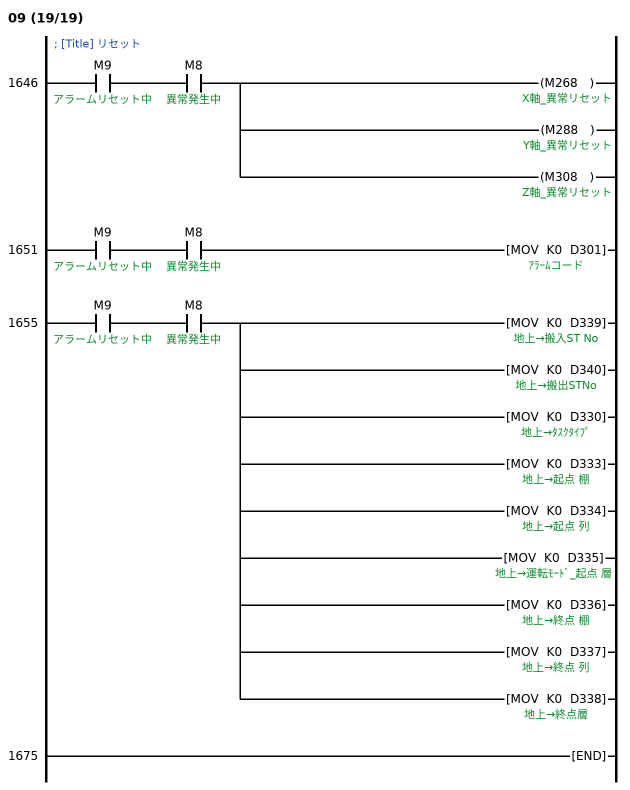
; [Title] リセット
1646  LD      M9  ; アラームリセット中
      AND     M8  ; 異常発生中
      OUT     M268  ; X軸_異常リセット
      OUT     M288  ; Y軸_異常リセット
      OUT     M308  ; Z軸_異常リセット
1651  LD      M9  ; アラームリセット中
      AND     M8  ; 異常発生中
      MOV     K0 D301
1655  LD      M9  ; アラームリセット中
      AND     M8  ; 異常発生中
      MOV     K0 D339  ; 地上→搬入ST No
      MOV     K0 D340  ; 地上→搬出STNo
      MOV     K0 D330
      MOV     K0 D333
      MOV     K0 D334
      MOV     K0 D335
      MOV     K0 D336
      MOV     K0 D337
      MOV     K0 D338
1675  END
END_PROGRAM

PROGRAM 10  // MAIN
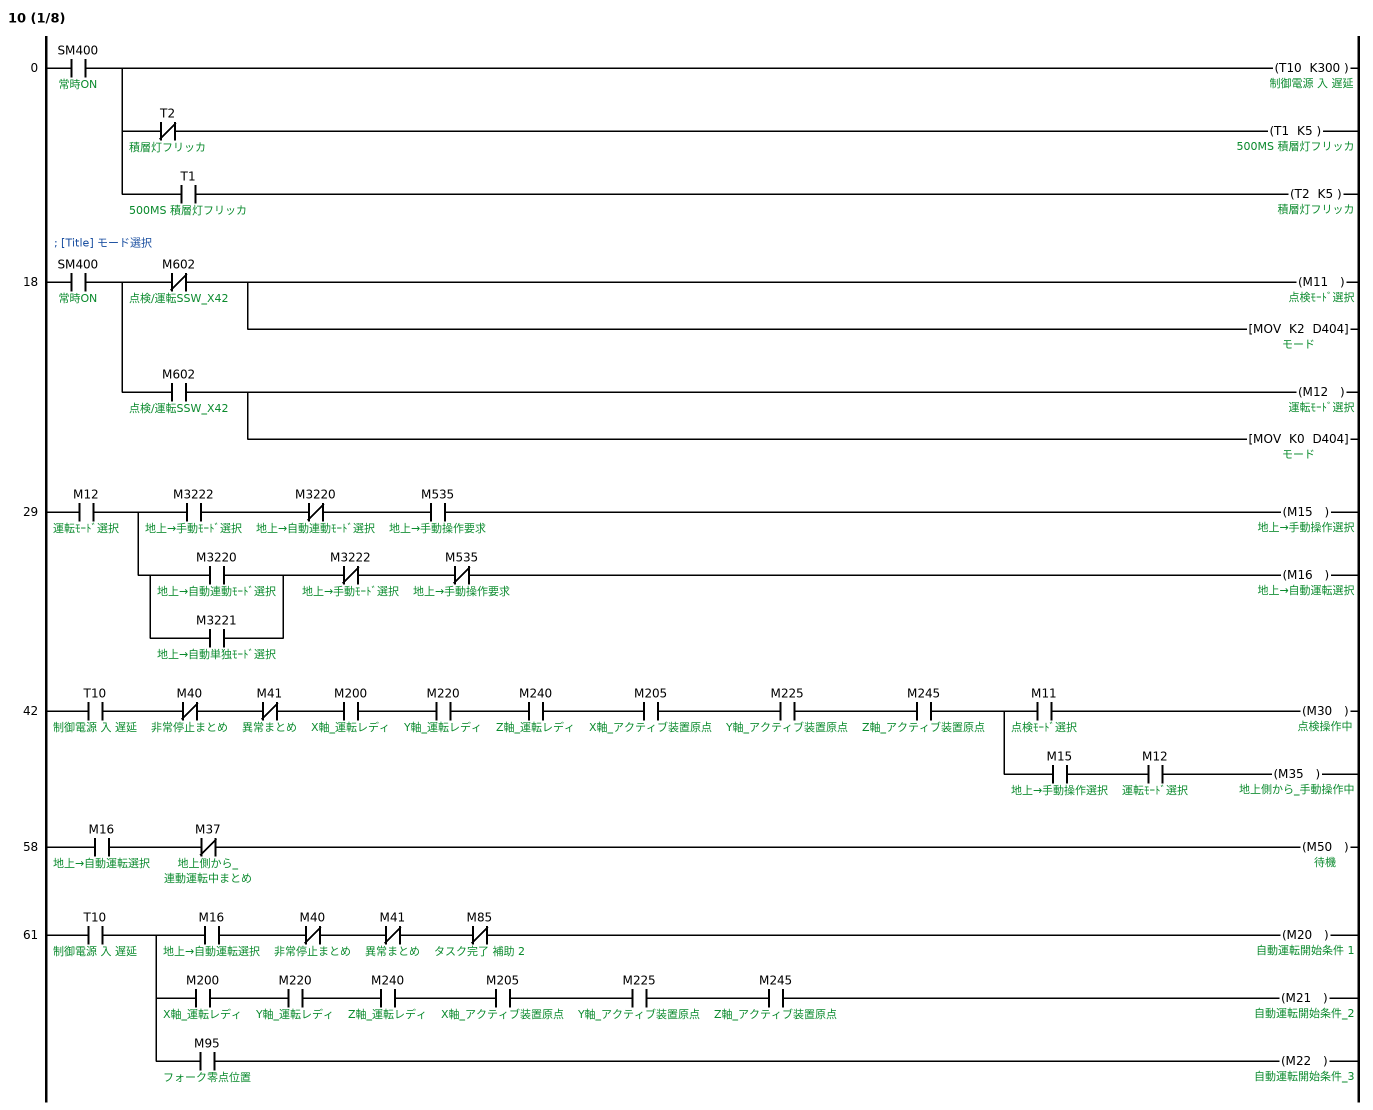
0     LD      SM400  ; 常時ON
      OUT     T10 K300  ; 制御電源 入 遅延
      MPS
      ANI     T2  ; 積層灯フリッカ
      OUT     T1 K5  ; 500MS 積層灯フリッカ
      MPP
      AND     T1  ; 500MS 積層灯フリッカ
      OUT     T2 K5  ; 積層灯フリッカ
; [Title] モード選択
18    LD      SM400  ; 常時ON
      MPS
      ANI     M602  ; 点検/運転SSW_X42
      OUT     M11  ; 点検ﾓｰﾄﾞ選択
      MOV     K2 D404  ; モード
      MPP
      AND     M602  ; 点検/運転SSW_X42
      OUT     M12  ; 運転ﾓｰﾄﾞ選択
      MOV     K0 D404
29    LD      M12  ; 運転ﾓｰﾄﾞ選択
      MPS
      AND     M3222  ; 地上→手動ﾓｰﾄﾞ選択
      ANI     M3220  ; 地上→自動連動ﾓｰﾄﾞ選択
      AND     M535  ; 地上→手動操作要求
      OUT     M15  ; 地上→手動操作選択
      MPP
      LD      M3220  ; 地上→自動連動ﾓｰﾄﾞ選択
      OR      M3221  ; 地上→自動単独ﾓｰﾄﾞ選択
      ANB
      ANI     M3222  ; 地上→手動ﾓｰﾄﾞ選択
      ANI     M535  ; 地上→手動操作要求
      OUT     M16  ; 地上→自動運転選択
42    LD      T10  ; 制御電源 入 遅延
      ANI     M40  ; 非常停止まとめ
      ANI     M41  ; 異常まとめ
      AND     M200  ; X軸_運転レディ
      AND     M220  ; Y軸_運転レディ
      AND     M240  ; Z軸_運転レディ
      AND     M205  ; X軸_アクティブ装置原点
      AND     M225  ; Y軸_アクティブ装置原点
      AND     M245  ; Z軸_アクティブ装置原点
      MPS
      AND     M11  ; 点検ﾓｰﾄﾞ選択
      OUT     M30  ; 点検操作中
      MPP
      AND     M15  ; 地上→手動操作選択
      AND     M12  ; 運転ﾓｰﾄﾞ選択
      OUT     M35  ; 地上側から_手動操作中
58    LD      M16  ; 地上→自動運転選択
      ANI     M37  ; 地上側から_連動運転中まとめ
      OUT     M50  ; 待機
61    LD      T10  ; 制御電源 入 遅延
      MPS
      AND     M16  ; 地上→自動運転選択
      ANI     M40  ; 非常停止まとめ
      ANI     M41  ; 異常まとめ
      ANI     M85  ; タスク完了 補助 2
      OUT     M20  ; 自動運転開始条件 1
      MRD
      AND     M200  ; X軸_運転レディ
      AND     M220  ; Y軸_運転レディ
      AND     M240  ; Z軸_運転レディ
      AND     M205  ; X軸_アクティブ装置原点
      AND     M225  ; Y軸_アクティブ装置原点
      AND     M245  ; Z軸_アクティブ装置原点
      OUT     M21  ; 自動運転開始条件_2
      MPP
      AND     M95  ; フォーク零点位置
      OUT     M22  ; 自動運転開始条件_3
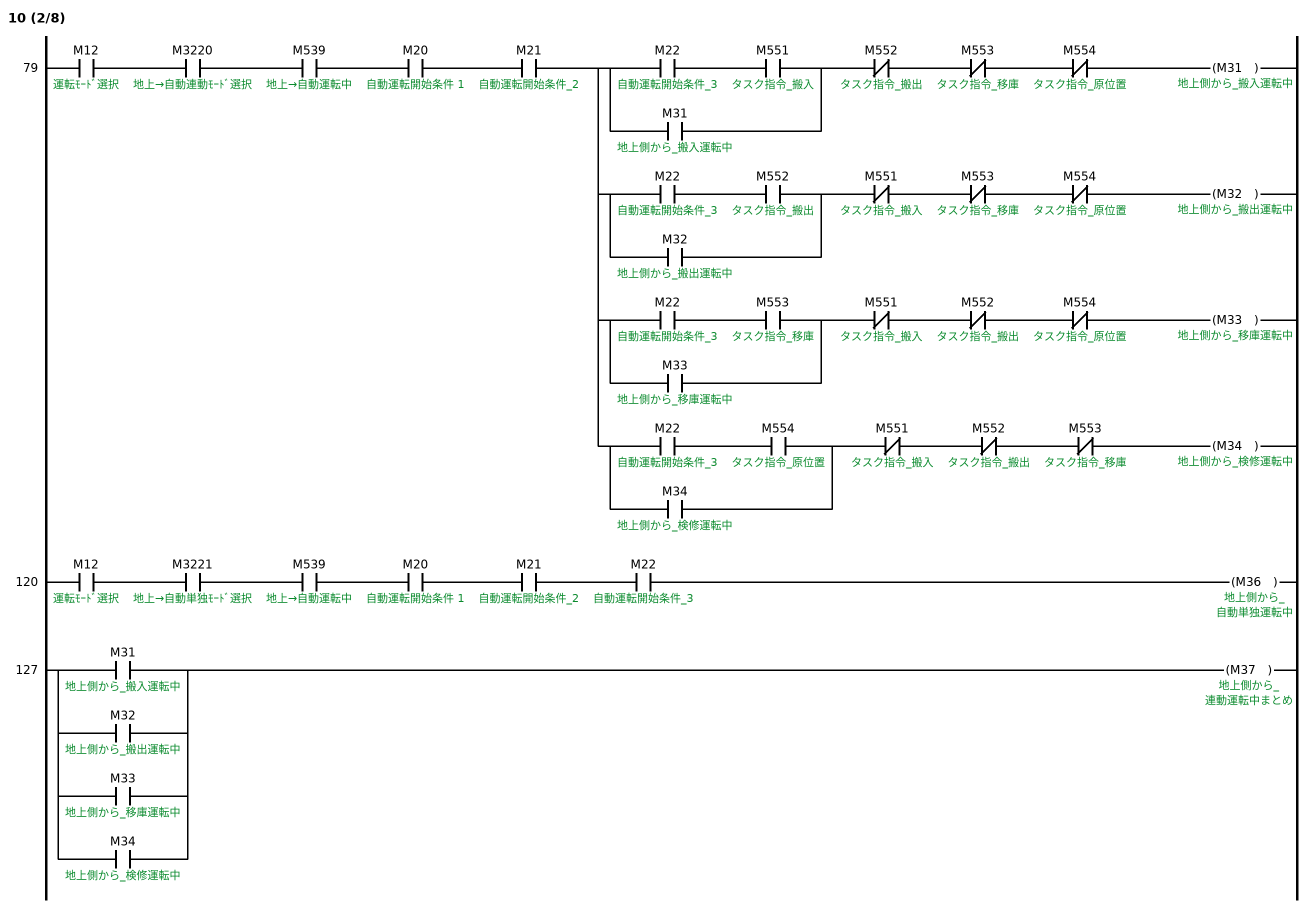
79    LD      M12  ; 運転ﾓｰﾄﾞ選択
      AND     M3220  ; 地上→自動連動ﾓｰﾄﾞ選択
      AND     M539  ; 地上→自動運転中
      AND     M20  ; 自動運転開始条件 1
      AND     M21  ; 自動運転開始条件_2
      MPS
      LD      M22  ; 自動運転開始条件_3
      AND     M551  ; タスク指令_搬入
      OR      M31  ; 地上側から_搬入運転中
      ANB
      ANI     M552  ; タスク指令_搬出
      ANI     M553  ; タスク指令_移庫
      ANI     M554  ; タスク指令_原位置
      OUT     M31  ; 地上側から_搬入運転中
      MRD
      LD      M22  ; 自動運転開始条件_3
      AND     M552  ; タスク指令_搬出
      OR      M32  ; 地上側から_搬出運転中
      ANB
      ANI     M551  ; タスク指令_搬入
      ANI     M553  ; タスク指令_移庫
      ANI     M554  ; タスク指令_原位置
      OUT     M32  ; 地上側から_搬出運転中
      MRD
      LD      M22  ; 自動運転開始条件_3
      AND     M553  ; タスク指令_移庫
      OR      M33  ; 地上側から_移庫運転中
      ANB
      ANI     M551  ; タスク指令_搬入
      ANI     M552  ; タスク指令_搬出
      ANI     M554  ; タスク指令_原位置
      OUT     M33  ; 地上側から_移庫運転中
      MPP
      LD      M22  ; 自動運転開始条件_3
      AND     M554  ; タスク指令_原位置
      OR      M34  ; 地上側から_検修運転中
      ANB
      ANI     M551  ; タスク指令_搬入
      ANI     M552  ; タスク指令_搬出
      ANI     M553  ; タスク指令_移庫
      OUT     M34  ; 地上側から_検修運転中
120   LD      M12  ; 運転ﾓｰﾄﾞ選択
      AND     M3221  ; 地上→自動単独ﾓｰﾄﾞ選択
      AND     M539  ; 地上→自動運転中
      AND     M20  ; 自動運転開始条件 1
      AND     M21  ; 自動運転開始条件_2
      AND     M22  ; 自動運転開始条件_3
      OUT     M36  ; 地上側から_自動単独運転中
127   LD      M31  ; 地上側から_搬入運転中
      OR      M32  ; 地上側から_搬出運転中
      OR      M33  ; 地上側から_移庫運転中
      OR      M34  ; 地上側から_検修運転中
      OUT     M37  ; 地上側から_連動運転中まとめ
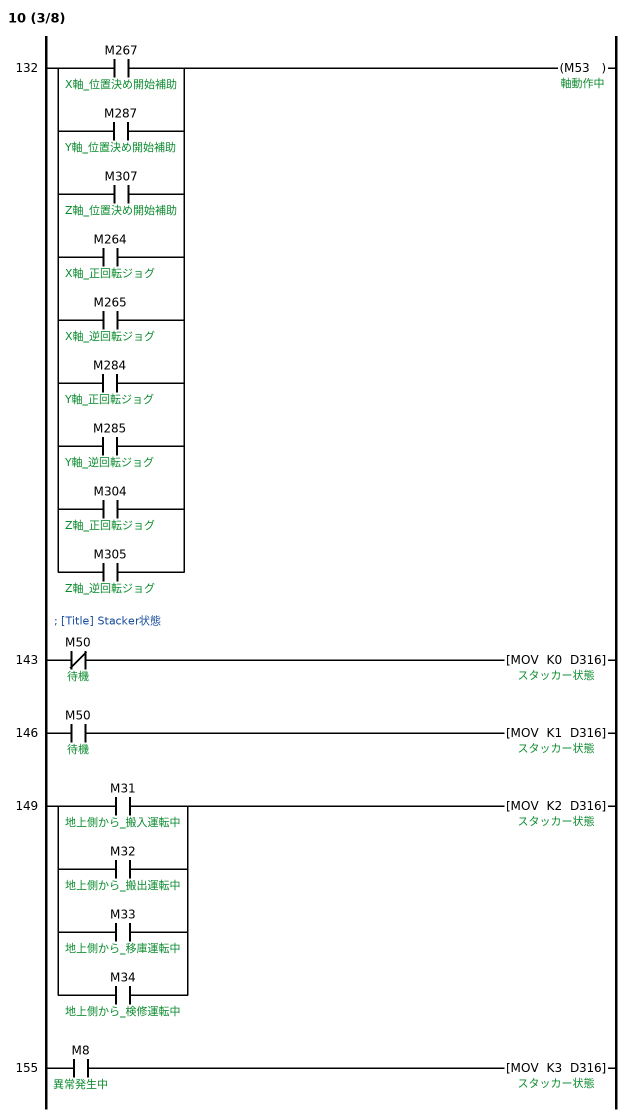
132   LD      M267  ; X軸_位置決め開始補助
      OR      M287  ; Y軸_位置決め開始補助
      OR      M307  ; Z軸_位置決め開始補助
      OR      M264  ; X軸_正回転ジョグ
      OR      M265  ; X軸_逆回転ジョグ
      OR      M284  ; Y軸_正回転ジョグ
      OR      M285  ; Y軸_逆回転ジョグ
      OR      M304  ; Z軸_正回転ジョグ
      OR      M305  ; Z軸_逆回転ジョグ
      OUT     M53  ; 軸動作中
; [Title] Stacker状態
143   LDI     M50  ; 待機
      MOV     K0 D316  ; スタッカー状態
146   LD      M50  ; 待機
      MOV     K1 D316
149   LD      M31  ; 地上側から_搬入運転中
      OR      M32  ; 地上側から_搬出運転中
      OR      M33  ; 地上側から_移庫運転中
      OR      M34  ; 地上側から_検修運転中
      MOV     K2 D316
155   LD      M8  ; 異常発生中
      MOV     K3 D316
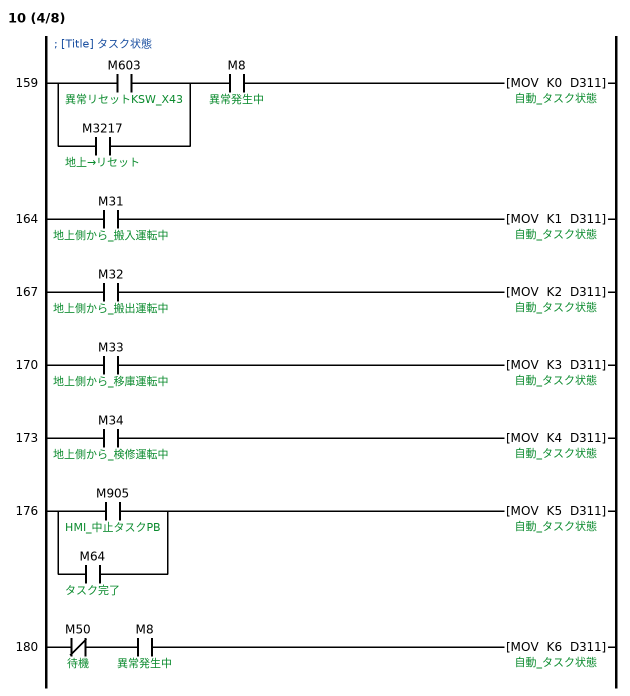
; [Title] タスク状態
159   LD      M603  ; 異常リセットKSW_X43
      OR      M3217  ; 地上→リセット
      AND     M8  ; 異常発生中
      MOV     K0 D311  ; 自動_タスク状態
164   LD      M31  ; 地上側から_搬入運転中
      MOV     K1 D311
167   LD      M32  ; 地上側から_搬出運転中
      MOV     K2 D311
170   LD      M33  ; 地上側から_移庫運転中
      MOV     K3 D311
173   LD      M34  ; 地上側から_検修運転中
      MOV     K4 D311
176   LD      M905  ; HMI_中止タスクPB
      OR      M64  ; タスク完了
      MOV     K5 D311
180   LDI     M50  ; 待機
      AND     M8  ; 異常発生中
      MOV     K6 D311
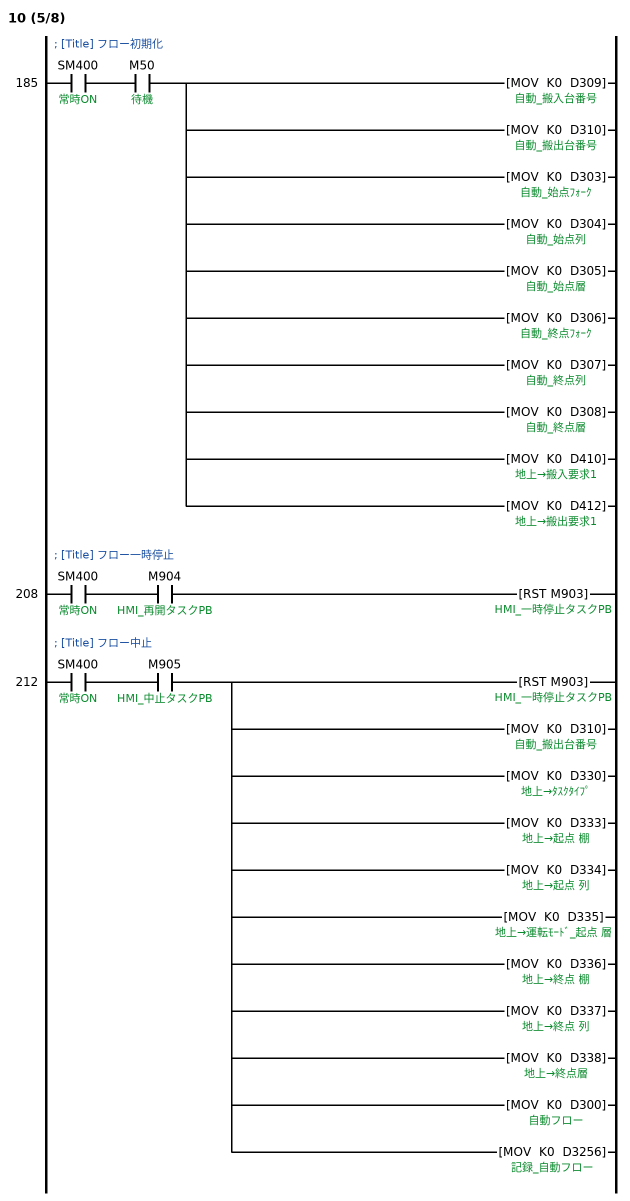
; [Title] フロー初期化
185   LD      SM400  ; 常時ON
      AND     M50  ; 待機
      MOV     K0 D309  ; 自動_搬入台番号
      MOV     K0 D310  ; 自動_搬出台番号
      MOV     K0 D303  ; 自動_始点ﾌｫｰｸ
      MOV     K0 D304  ; 自動_始点列
      MOV     K0 D305  ; 自動_始点層
      MOV     K0 D306  ; 自動_終点ﾌｫｰｸ
      MOV     K0 D307  ; 自動_終点列
      MOV     K0 D308  ; 自動_終点層
      MOV     K0 D410  ; 地上→搬入要求1
      MOV     K0 D412  ; 地上→搬出要求1
; [Title] フロー一時停止
208   LD      SM400  ; 常時ON
      AND     M904  ; HMI_再開タスクPB
      RST     M903  ; HMI_一時停止タスクPB
; [Title] フロー中止
212   LD      SM400  ; 常時ON
      AND     M905  ; HMI_中止タスクPB
      RST     M903  ; HMI_一時停止タスクPB
      MOV     K0 D310
      MOV     K0 D330  ; 地上→ﾀｽｸﾀｲﾌﾟ
      MOV     K0 D333  ; 地上→起点 棚
      MOV     K0 D334  ; 地上→起点 列
      MOV     K0 D335  ; 地上→運転ﾓｰﾄﾞ_起点 層
      MOV     K0 D336  ; 地上→終点 棚
      MOV     K0 D337  ; 地上→終点 列
      MOV     K0 D338  ; 地上→終点層
      MOV     K0 D300  ; 自動フロー
      MOV     K0 D3256  ; 記録_自動フロー
